	#index := #index + 1;
	//++++++++++++++++++++++++++++++++++++++++++++++++++++++++++++++/*276*/
	"DB_BIBLIOTHEQUE".Mobile[#index].Nom := 'BDE10';
	"DB_BIBLIOTHEQUE".Mobile[#index].Noeud := TRUE;
	"DB_BIBLIOTHEQUE".Mobile[#index].Mob_Suiv[0] := "Index_Mobile"('BB01');
	"DB_BIBLIOTHEQUE".Mobile[#index].Mob_Suiv[1] := "Index_Mobile"('BB02');
	"DB_BIBLIOTHEQUE".Mobile[#index].Pos[0].Nom := 'DROITE';
	"DB_BIBLIOTHEQUE".Mobile[#index].Pos[0].Mob_Suiv[0] := "Index_Mobile"('BB02');
	"DB_BIBLIOTHEQUE".Mobile[#index].Pos[1].Nom := 'GAUCHE';
	"DB_BIBLIOTHEQUE".Mobile[#index].Pos[1].Mob_Suiv[0] := "Index_Mobile"('BB01');
	"Init_Tps"(#index);


	//Entrées
	"DB_BIBLIOTHEQUE".Mobile[#index].Pos[0].Entr0_Ap_Pos[0] := "I_RP_BDE10_BB1";
	"DB_BIBLIOTHEQUE".Mobile[#index].Pos[0].Entr1_Ap_Pos[0] := "I_RP_BDE10_BB2";
	// "DB_BIBLIOTHEQUE".Mobile[#index].Pos[0].Sort1[0] := "I_CP_B2DE10_BB2";
	// "DB_BIBLIOTHEQUE".Mobile[#index].Pos[0].Sort0[0] := "I_CP_B2DE10_BB1";
	// "DB_BIBLIOTHEQUE".Mobile[#index].Pos[0].Sort0_Pr_Fin_Pos[0] := "I_CP_B2DE10_BB2";
	// "DB_BIBLIOTHEQUE".Mobile[#index].Pos[0].Sort0_Pr_Fin_Pos[1] := "I_CP_B2DE10_BB1";

	"DB_BIBLIOTHEQUE".Mobile[#index].Pos[1].Entr0_Ap_Pos[1] := "I_RP_BDE10_BB2";
	"DB_BIBLIOTHEQUE".Mobile[#index].Pos[1].Entr1_Ap_Pos[0] := "I_RP_BDE10_BB1";

	//Sorties
	// "DB_BIBLIOTHEQUE".Mobile[#index].Pos[1].Sort1[0] := "I_CP_B2DE10_BB1";
	// "DB_BIBLIOTHEQUE".Mobile[#index].Pos[1].Sort0[0] := "I_CP_B2DE10_BB2";
	// "DB_BIBLIOTHEQUE".Mobile[#index].Pos[1].Sort0_Pr_Fin_Pos[0] := "I_CP_B2DE10_BB2";
	// "DB_BIBLIOTHEQUE".Mobile[#index].Pos[1].Sort0_Pr_Fin_Pos[1] := "I_CP_B2DE10_BB1";
	#index := #index + 1;
	//++++++++++++++++++++++++++++++++++++++++++++++++++++++++++++++/*277*/
	"DB_BIBLIOTHEQUE".Mobile[#index].Nom := 'E11';
	"DB_BIBLIOTHEQUE".Mobile[#index].Mob_Suiv[0] := "Index_Mobile"('BDE11');
	"DB_BIBLIOTHEQUE".Mobile[#index].Pos[0].Nom := 'DROIT';
	"DB_BIBLIOTHEQUE".Mobile[#index].Pos[0].Mob_Suiv[0] := "Index_Mobile"('BDE11');
	"Init_Tps"(#index);

	// Entrées avant pos
	"DB_BIBLIOTHEQUE".Mobile[#index].Pos[0].Entr0_Av_Pos[0] := "I_RD_DISJ_E11";
	"DB_BIBLIOTHEQUE".Mobile[#index].Pos[0].Entr0_Av_Pos[1] := "I_RD_DBHG_E11";
	"DB_BIBLIOTHEQUE".Mobile[#index].Pos[0].Entr0_Av_Pos[2] := "I_RD_DBHD_E11";
	"DB_BIBLIOTHEQUE".Mobile[#index].Pos[0].Entr0_Av_Pos[3] := "I_RD_DBBG_E11";
	"DB_BIBLIOTHEQUE".Mobile[#index].Pos[0].Entr0_Av_Pos[4] := "I_RD_DBBD_E11";
	// Entrées apres pos
	"DB_BIBLIOTHEQUE".Mobile[#index].Pos[0].Entr0_Ap_Pos[0] := "I_RD_DISJ_E11";
	"DB_BIBLIOTHEQUE".Mobile[#index].Pos[0].Entr0_Ap_Pos[1] := "I_RD_DBHG_E11";
	"DB_BIBLIOTHEQUE".Mobile[#index].Pos[0].Entr0_Ap_Pos[2] := "I_RD_DBHD_E11";
	"DB_BIBLIOTHEQUE".Mobile[#index].Pos[0].Entr0_Ap_Pos[3] := "I_RD_DBBG_E11";
	"DB_BIBLIOTHEQUE".Mobile[#index].Pos[0].Entr0_Ap_Pos[4] := "I_RD_DBBD_E11";

	"DB_BIBLIOTHEQUE".Mobile[#index].Pos[0].Entr1_Ap_Pos[0] := "I_RR_E11";
	"DB_BIBLIOTHEQUE".Mobile[#index].Pos[0].Entr1_Ap_Pos[1] := "I_RM_E11";


	// Entrées fin pos
	"DB_BIBLIOTHEQUE".Mobile[#index].Pos[0].Entr0_Ap_Fin_Pos[0] := "I_RM_E11";

	// Sorties
	"DB_BIBLIOTHEQUE".Mobile[#index].Pos[0].Sort1[0] := "I_CM_E11";
	"DB_BIBLIOTHEQUE".Mobile[#index].Pos[0].Sort0_Pr_Fin_Pos[0] := "I_CM_E11";
	#index := #index + 1;
	//++++++++++++++++++++++++++++++++++++++++++++++++++++++++++++++/*278*/
	"DB_BIBLIOTHEQUE".Mobile[#index].Nom := 'BDE11';
	"DB_BIBLIOTHEQUE".Mobile[#index].Noeud := TRUE;
	"DB_BIBLIOTHEQUE".Mobile[#index].Mob_Suiv[0] := "Index_Mobile"('TMEL');
	"DB_BIBLIOTHEQUE".Mobile[#index].Mob_Suiv[1] := "Index_Mobile"('TMEL2');
	"DB_BIBLIOTHEQUE".Mobile[#index].Pos[0].Nom := 'DROITE';
	"DB_BIBLIOTHEQUE".Mobile[#index].Pos[0].Mob_Suiv[0] := "Index_Mobile"('TMEL');
	"DB_BIBLIOTHEQUE".Mobile[#index].Pos[1].Nom := 'GAUCHE';
	"DB_BIBLIOTHEQUE".Mobile[#index].Pos[1].Mob_Suiv[0] := "Index_Mobile"('TMEL2');


	"Init_Tps"(#index);

	//Entrées
	"DB_BIBLIOTHEQUE".Mobile[#index].Pos[0].Entr0_Ap_Pos[0] := "I_RP_BDE11_TMEL2";
	"DB_BIBLIOTHEQUE".Mobile[#index].Pos[0].Entr1_Ap_Pos[0] := "I_RP_BDE11_TMEL1";
	"DB_BIBLIOTHEQUE".Mobile[#index].Pos[0].Sort1[0] := "I_CP_BDE11_TMEL1";
	"DB_BIBLIOTHEQUE".Mobile[#index].Pos[0].Sort0[0] := "I_CP_BDE11_TMEL2";
	"DB_BIBLIOTHEQUE".Mobile[#index].Pos[0].Sort0_Pr_Fin_Pos[0] := "I_CP_BDE11_TMEL1";
	"DB_BIBLIOTHEQUE".Mobile[#index].Pos[0].Sort0_Pr_Fin_Pos[1] := "I_CP_BDE11_TMEL2";


	"DB_BIBLIOTHEQUE".Mobile[#index].Pos[1].Entr0_Ap_Pos[1] := "I_RP_BDE11_TMEL1";
	"DB_BIBLIOTHEQUE".Mobile[#index].Pos[1].Entr1_Ap_Pos[0] := "I_RP_BDE11_TMEL2";

	//Sorties
	"DB_BIBLIOTHEQUE".Mobile[#index].Pos[1].Sort1[0] := "I_CP_BDE11_TMEL2";
	"DB_BIBLIOTHEQUE".Mobile[#index].Pos[1].Sort0[0] := "I_CP_BDE11_TMEL1";
	"DB_BIBLIOTHEQUE".Mobile[#index].Pos[1].Sort0_Pr_Fin_Pos[0] := "I_CP_BDE11_TMEL1";
	"DB_BIBLIOTHEQUE".Mobile[#index].Pos[1].Sort0_Pr_Fin_Pos[1] := "I_CP_BDE11_TMEL2";
	#index := #index + 1;
	//++++++++++++++++++++++++++++++++++++++++++++++++++++++++++++++/*279*/
	"DB_BIBLIOTHEQUE".Mobile[#index].Nom := 'E30';
	"DB_BIBLIOTHEQUE".Mobile[#index].Mob_Suiv[0] := "Index_Mobile"('T20');
	"DB_BIBLIOTHEQUE".Mobile[#index].Pos[0].Nom := 'MARCHE';
	"DB_BIBLIOTHEQUE".Mobile[#index].Pos[0].Mob_Suiv[0] := "Index_Mobile"('T20');
	"DB_BIBLIOTHEQUE".Mobile[#index].Tps_Asserv := t#3s;
	"DB_BIBLIOTHEQUE".Mobile[#index].Tps_Vid := t#3s;
	"DB_BIBLIOTHEQUE".Mobile[#index].Tps_Att := t#500ms;
	"DB_BIBLIOTHEQUE".Mobile[#index].Tps_Arr := t#0ms;
	"DB_BIBLIOTHEQUE".Mobile[#index].Tps_Max_Mar_Forc := t#5s;

	// Entrées avant pos
	"DB_BIBLIOTHEQUE".Mobile[#index].Pos[0].Entr0_Av_Pos[0] := "I_RD_DISJ_E30";
	"DB_BIBLIOTHEQUE".Mobile[#index].Pos[0].Entr0_Av_Pos[1] := "I_RD_DBHG_E30";
	"DB_BIBLIOTHEQUE".Mobile[#index].Pos[0].Entr0_Av_Pos[2] := "I_RD_DBHD_E30";
	"DB_BIBLIOTHEQUE".Mobile[#index].Pos[0].Entr0_Av_Pos[3] := "I_RD_DBBG_E30";
	"DB_BIBLIOTHEQUE".Mobile[#index].Pos[0].Entr0_Av_Pos[4] := "I_RD_DBBD_E30";
	// Entrées apres pos
	"DB_BIBLIOTHEQUE".Mobile[#index].Pos[0].Entr0_Ap_Pos[0] := "I_RD_DISJ_E30";
	"DB_BIBLIOTHEQUE".Mobile[#index].Pos[0].Entr0_Ap_Pos[1] := "I_RD_DBHG_E30";
	"DB_BIBLIOTHEQUE".Mobile[#index].Pos[0].Entr0_Ap_Pos[2] := "I_RD_DBHD_E30";
	"DB_BIBLIOTHEQUE".Mobile[#index].Pos[0].Entr0_Ap_Pos[3] := "I_RD_DBBG_E30";
	"DB_BIBLIOTHEQUE".Mobile[#index].Pos[0].Entr0_Ap_Pos[4] := "I_RD_DBBD_E30";

	// "DB_BIBLIOTHEQUE".Mobile[#index].Pos[0].Entr1_Ap_Pos[0] := "I_RR_E30";
	"DB_BIBLIOTHEQUE".Mobile[#index].Pos[0].Entr1_Ap_Pos[0] := "I_RM_E30";


	// Entrées fin pos
	//"DB_BIBLIOTHEQUE".Mobile[#index].Pos[0].Entr0_Ap_Fin_Pos[0]:="I_RM_E30";

	// Sorties
	"DB_BIBLIOTHEQUE".Mobile[#index].Pos[0].Sort1[0] := "I_CM_E30";
	"DB_BIBLIOTHEQUE".Mobile[#index].Pos[0].Sort0_Pr_Fin_Pos[0] := "I_CM_E30";
	#index := #index + 1;
	//++++++++++++++++++++++++++++++++++++++++++++++++++++++++++++++/*280*/
	"DB_BIBLIOTHEQUE".Mobile[#index].Nom := 'Ext1_BB1';
	"DB_BIBLIOTHEQUE".Mobile[#index].Pos[0].Nom := 'FERMETURE';
	"DB_BIBLIOTHEQUE".Mobile[#index].Pos[1].Nom := 'OUVERTURE';
	"DB_BIBLIOTHEQUE".Mobile[#index].Tjr_Desasservi := TRUE;
	"Init_Tps"(#index);

	//position fermeture
	"DB_BIBLIOTHEQUE".Mobile[#index].Pos[0].Entr0_Ap_Pos[0] := "I_RPO_TRBB1";
	"DB_BIBLIOTHEQUE".Mobile[#index].Pos[0].Entr1_Ap_Pos[0] := "I_RPF_TRBB1";
	"DB_BIBLIOTHEQUE".Mobile[#index].Pos[0].Sort0[0] := "I_CO_TRBB1";
	"DB_BIBLIOTHEQUE".Mobile[#index].Pos[0].Sort0_Pr_Fin_Pos[0] := "I_CO_TRBB1";

	//position ouverture
	"DB_BIBLIOTHEQUE".Mobile[#index].Pos[1].Entr0_Ap_Pos[0] := "I_RPF_TRBB1";
	"DB_BIBLIOTHEQUE".Mobile[#index].Pos[1].Entr1_Ap_Pos[0] := "I_RPO_TRBB1";
	"DB_BIBLIOTHEQUE".Mobile[#index].Pos[1].Sort1[0] := "I_CO_TRBB1";
	"DB_BIBLIOTHEQUE".Mobile[#index].Pos[1].Sort0_Pr_Fin_Pos[0] := "I_CO_TRBB1";
	#index := #index + 1;
	//++++++++++++++++++++++++++++++++++++++++++++++++++++++++++++++/*281*/
	"DB_BIBLIOTHEQUE".Mobile[#index].Nom := 'Ext1_BB2';
	"DB_BIBLIOTHEQUE".Mobile[#index].Pos[0].Nom := 'FERMETURE';
	"DB_BIBLIOTHEQUE".Mobile[#index].Pos[1].Nom := 'OUVERTURE';
	"DB_BIBLIOTHEQUE".Mobile[#index].Tjr_Desasservi := TRUE;
	"Init_Tps"(#index);

	//position fermeture
	"DB_BIBLIOTHEQUE".Mobile[#index].Pos[0].Entr0_Ap_Pos[0] := "I_RPO_TRBB2";
	"DB_BIBLIOTHEQUE".Mobile[#index].Pos[0].Entr1_Ap_Pos[0] := "I_RPF_TRBB2";
	"DB_BIBLIOTHEQUE".Mobile[#index].Pos[0].Sort0[0] := "I_CO_TRBB2";
	"DB_BIBLIOTHEQUE".Mobile[#index].Pos[0].Sort0_Pr_Fin_Pos[0] := "I_CO_TRBB2";

	//position ouverture
	"DB_BIBLIOTHEQUE".Mobile[#index].Pos[1].Entr0_Ap_Pos[0] := "I_RPF_TRBB2";
	"DB_BIBLIOTHEQUE".Mobile[#index].Pos[1].Entr1_Ap_Pos[0] := "I_RPO_TRBB2";
	"DB_BIBLIOTHEQUE".Mobile[#index].Pos[1].Sort1[0] := "I_CO_TRBB2";
	"DB_BIBLIOTHEQUE".Mobile[#index].Pos[1].Sort0_Pr_Fin_Pos[0] := "I_CO_TRBB2";
	#index := #index + 1;
	//++++++++++++++++++++++++++++++++++++++++++++++++++++++++++++++/*282*/
	"DB_BIBLIOTHEQUE".Mobile[#index].Nom := 'Ext1_S50';
	"DB_BIBLIOTHEQUE".Mobile[#index].Mob_Suiv[0] := "Index_Mobile"('EXT2_S50');
	"Init_Tps"(#index);

	// Position PV
	"DB_BIBLIOTHEQUE".Mobile[#index].Pos[0].Nom := 'MARCHE_PV';
	"DB_BIBLIOTHEQUE".Mobile[#index].Pos[0].Mob_Suiv[0] := "Index_Mobile"('EXT2_S50');
	"DB_BIBLIOTHEQUE".Mobile[#index].Pos[0].Suiv_Enc := "Index_Mobile"('EXT2_S50');

	// Entrées avant pos
	"DB_BIBLIOTHEQUE".Mobile[#index].Pos[0].Entr0_Av_Pos[0] := "I_RD_DISJ_EXT1_S50";
	// "DB_BIBLIOTHEQUE".Mobile[#index].Pos[0].Entr0_Av_Pos[1] := "I_RD_VFD_BP4";

	// Entrées apres pos
	"DB_BIBLIOTHEQUE".Mobile[#index].Pos[0].Entr0_Ap_Pos[1] := "I_RD_DISJ_EXT1_S50";
	//"DB_BIBLIOTHEQUE".Mobile[#index].Pos[0].Entr0_Ap_Pos[2] := "I_RD_VFD_BP4";
	//"DB_BIBLIOTHEQUE".Mobile[#index].Pos[0].Entr1_Ap_Pos[0] := "I_RR_EXT1_S50";
	"DB_BIBLIOTHEQUE".Mobile[#index].Pos[0].Entr1_Ap_Pos[0] := "I_RM_EXT1_S50";

	// Entrées fin pos
	"DB_BIBLIOTHEQUE".Mobile[#index].Pos[0].Entr0_Ap_Fin_Pos[0] := "I_RM_EXT1_S50";

	// Sorties
	"DB_BIBLIOTHEQUE".Mobile[#index].Pos[0].Sort1[0] := "I_CM_EXT1_S50";
	"DB_BIBLIOTHEQUE".Mobile[#index].Pos[0].Sort1[1] := "I_CPV_SBP4";
	"DB_BIBLIOTHEQUE".Mobile[#index].Pos[0].Sort0_Pr_Fin_Pos[0] := "I_CM_EXT1_S50";
	"DB_BIBLIOTHEQUE".Mobile[#index].Pos[0].Sort0_Pr_Fin_Pos[1] := "I_CPV_SBP4";

	// Position GV
	"DB_BIBLIOTHEQUE".Mobile[#index].Pos[1].Nom := 'MARCHE_GV';
	"DB_BIBLIOTHEQUE".Mobile[#index].Pos[1].Mob_Suiv[0] := "Index_Mobile"('EXT2_S50');
	"DB_BIBLIOTHEQUE".Mobile[#index].Pos[1].Suiv_Enc := "Index_Mobile"('EXT2_S50');

	// Entrées avant pos
	"DB_BIBLIOTHEQUE".Mobile[#index].Pos[1].Entr0_Av_Pos[0] := "I_RD_DISJ_EXT1_S50";
	// "DB_BIBLIOTHEQUE".Mobile[#index].Pos[0].Entr0_Av_Pos[1] := "I_RD_VFD_BP4";

	// Entrées apres pos
	"DB_BIBLIOTHEQUE".Mobile[#index].Pos[1].Entr0_Ap_Pos[1] := "I_RD_DISJ_EXT1_S50";
	//"DB_BIBLIOTHEQUE".Mobile[#index].Pos[0].Entr0_Ap_Pos[2] := "I_RD_VFD_BP4";
	//"DB_BIBLIOTHEQUE".Mobile[#index].Pos[0].Entr1_Ap_Pos[0] := "I_RR_EXT1_S50";
	"DB_BIBLIOTHEQUE".Mobile[#index].Pos[1].Entr1_Ap_Pos[0] := "I_RM_EXT1_S50";

	// Entrées fin pos
	"DB_BIBLIOTHEQUE".Mobile[#index].Pos[1].Entr0_Ap_Fin_Pos[0] := "I_RM_EXT1_S50";

	// Sorties
	"DB_BIBLIOTHEQUE".Mobile[#index].Pos[1].Sort1[0] := "I_CM_EXT1_S50";
	"DB_BIBLIOTHEQUE".Mobile[#index].Pos[1].Sort1[1] := "I_CGV_SBP4";
	"DB_BIBLIOTHEQUE".Mobile[#index].Pos[1].Sort0_Pr_Fin_Pos[0] := "I_CM_EXT1_S50";
	"DB_BIBLIOTHEQUE".Mobile[#index].Pos[1].Sort0_Pr_Fin_Pos[1] := "I_CGV_SBP4";
	#index := #index + 1;
	//++++++++++++++++++++++++++++++++++++++++++++++++++++++++++++++/*283*/
	"DB_BIBLIOTHEQUE".Mobile[#index].Nom := 'Ext1_S51';
	"DB_BIBLIOTHEQUE".Mobile[#index].Mob_Suiv[0] := "Index_Mobile"('EXT2_S51');
	"Init_Tps"(#index);

	// Position PV
	"DB_BIBLIOTHEQUE".Mobile[#index].Pos[0].Nom := 'MARCHE_PV';
	"DB_BIBLIOTHEQUE".Mobile[#index].Pos[0].Mob_Suiv[0] := "Index_Mobile"('EXT2_S51');
	"DB_BIBLIOTHEQUE".Mobile[#index].Pos[0].Suiv_Enc := "Index_Mobile"('EXT2_S51');
	// Entrées avant pos
	"DB_BIBLIOTHEQUE".Mobile[#index].Pos[0].Entr0_Av_Pos[0] := "I_RD_DISJ_EXT1_S51";
	//"DB_BIBLIOTHEQUE".Mobile[#index].Pos[0].Entr0_Av_Pos[1] := "I_RD_VFD_BP4";

	// Entrées apres pos
	"DB_BIBLIOTHEQUE".Mobile[#index].Pos[0].Entr0_Ap_Pos[1] := "I_RD_DISJ_EXT1_S51";
	//"DB_BIBLIOTHEQUE".Mobile[#index].Pos[0].Entr0_Ap_Pos[2] := "I_RD_VFD_BP4";
	//"DB_BIBLIOTHEQUE".Mobile[#index].Pos[0].Entr1_Ap_Pos[0] := "I_RR_EXT1_S51";
	"DB_BIBLIOTHEQUE".Mobile[#index].Pos[0].Entr1_Ap_Pos[0] := "I_RM_EXT1_S51";

	// Entrées fin pos
	"DB_BIBLIOTHEQUE".Mobile[#index].Pos[0].Entr0_Ap_Fin_Pos[0] := "I_RM_EXT1_S51";

	// Sorties
	"DB_BIBLIOTHEQUE".Mobile[#index].Pos[0].Sort1[0] := "I_CM_EXT1_S51";
	"DB_BIBLIOTHEQUE".Mobile[#index].Pos[0].Sort1[1] := "I_CPV_SBP4";
	"DB_BIBLIOTHEQUE".Mobile[#index].Pos[0].Sort0_Pr_Fin_Pos[0] := "I_CM_EXT1_S51";
	"DB_BIBLIOTHEQUE".Mobile[#index].Pos[0].Sort0_Pr_Fin_Pos[1] := "I_CPV_SBP4";

	// Position GV
	"DB_BIBLIOTHEQUE".Mobile[#index].Pos[1].Nom := 'MARCHE_GV';
	"DB_BIBLIOTHEQUE".Mobile[#index].Pos[1].Mob_Suiv[0] := "Index_Mobile"('EXT2_S51');
	"DB_BIBLIOTHEQUE".Mobile[#index].Pos[1].Suiv_Enc := "Index_Mobile"('EXT2_S51');
	// Entrées avant pos
	"DB_BIBLIOTHEQUE".Mobile[#index].Pos[1].Entr0_Av_Pos[0] := "I_RD_DISJ_EXT1_S51";
	//"DB_BIBLIOTHEQUE".Mobile[#index].Pos[0].Entr0_Av_Pos[1] := "I_RD_VFD_BP4";

	// Entrées apres pos
	"DB_BIBLIOTHEQUE".Mobile[#index].Pos[1].Entr0_Ap_Pos[1] := "I_RD_DISJ_EXT1_S51";
	//"DB_BIBLIOTHEQUE".Mobile[#index].Pos[0].Entr0_Ap_Pos[2] := "I_RD_VFD_BP4";
	//"DB_BIBLIOTHEQUE".Mobile[#index].Pos[0].Entr1_Ap_Pos[0] := "I_RR_EXT1_S51";
	"DB_BIBLIOTHEQUE".Mobile[#index].Pos[1].Entr1_Ap_Pos[0] := "I_RM_EXT1_S51";

	// Entrées fin pos
	"DB_BIBLIOTHEQUE".Mobile[#index].Pos[1].Entr0_Ap_Fin_Pos[0] := "I_RM_EXT1_S51";

	// Sorties
	"DB_BIBLIOTHEQUE".Mobile[#index].Pos[1].Sort1[0] := "I_CM_EXT1_S51";
	"DB_BIBLIOTHEQUE".Mobile[#index].Pos[1].Sort1[1] := "I_CGV_SBP4";
	"DB_BIBLIOTHEQUE".Mobile[#index].Pos[1].Sort0_Pr_Fin_Pos[0] := "I_CM_EXT1_S51";
	"DB_BIBLIOTHEQUE".Mobile[#index].Pos[1].Sort0_Pr_Fin_Pos[1] := "I_CGV_SBP4";
	#index := #index + 1;
	//++++++++++++++++++++++++++++++++++++++++++++++++++++++++++++++/*284*/
	"DB_BIBLIOTHEQUE".Mobile[#index].Nom := 'Ext1_S52';
	"DB_BIBLIOTHEQUE".Mobile[#index].Mob_Suiv[0] := "Index_Mobile"('EXT2_S52');
	"Init_Tps"(#index);

	// Position PV
	"DB_BIBLIOTHEQUE".Mobile[#index].Pos[0].Nom := 'MARCHE_PV';
	"DB_BIBLIOTHEQUE".Mobile[#index].Pos[0].Mob_Suiv[0] := "Index_Mobile"('EXT2_S52');
	"DB_BIBLIOTHEQUE".Mobile[#index].Pos[0].Suiv_Enc := "Index_Mobile"('EXT2_S52');
	// Entrées avant pos
	"DB_BIBLIOTHEQUE".Mobile[#index].Pos[0].Entr0_Av_Pos[0] := "I_RD_DISJ_EXT1_S52";
	//"DB_BIBLIOTHEQUE".Mobile[#index].Pos[0].Entr0_Av_Pos[1] := "I_RD_VFD_BP4";
	// Entrées apres pos

	"DB_BIBLIOTHEQUE".Mobile[#index].Pos[0].Entr0_Ap_Pos[1] := "I_RD_DISJ_EXT1_S52";
	//"DB_BIBLIOTHEQUE".Mobile[#index].Pos[0].Entr0_Ap_Pos[2] := "I_RD_VFD_BP4";

	//"DB_BIBLIOTHEQUE".Mobile[#index].Pos[0].Entr1_Ap_Pos[0] := "I_RR_EXT1_S52";
	"DB_BIBLIOTHEQUE".Mobile[#index].Pos[0].Entr1_Ap_Pos[0] := "I_RM_EXT1_S52";

	// Entrées fin pos
	"DB_BIBLIOTHEQUE".Mobile[#index].Pos[0].Entr0_Ap_Fin_Pos[0] := "I_RM_EXT1_S52";

	// Sorties
	"DB_BIBLIOTHEQUE".Mobile[#index].Pos[0].Sort1[0] := "I_CM_EXT1_S52";
	"DB_BIBLIOTHEQUE".Mobile[#index].Pos[0].Sort1[1] := "I_CPV_SBP4";
	"DB_BIBLIOTHEQUE".Mobile[#index].Pos[0].Sort0_Pr_Fin_Pos[0] := "I_CM_EXT1_S52";
	"DB_BIBLIOTHEQUE".Mobile[#index].Pos[0].Sort0_Pr_Fin_Pos[1] := "I_CPV_SBP4";

	// Position GV
	"DB_BIBLIOTHEQUE".Mobile[#index].Pos[1].Nom := 'MARCHE_GV';
	"DB_BIBLIOTHEQUE".Mobile[#index].Pos[1].Mob_Suiv[0] := "Index_Mobile"('EXT2_S52');
	"DB_BIBLIOTHEQUE".Mobile[#index].Pos[1].Suiv_Enc := "Index_Mobile"('EXT2_S52');
	// Entrées avant pos
	"DB_BIBLIOTHEQUE".Mobile[#index].Pos[1].Entr0_Av_Pos[0] := "I_RD_DISJ_EXT1_S52";
	//"DB_BIBLIOTHEQUE".Mobile[#index].Pos[0].Entr0_Av_Pos[1] := "I_RD_VFD_BP4";
	// Entrées apres pos

	"DB_BIBLIOTHEQUE".Mobile[#index].Pos[1].Entr0_Ap_Pos[1] := "I_RD_DISJ_EXT1_S52";
	//"DB_BIBLIOTHEQUE".Mobile[#index].Pos[0].Entr0_Ap_Pos[2] := "I_RD_VFD_BP4";

	//"DB_BIBLIOTHEQUE".Mobile[#index].Pos[0].Entr1_Ap_Pos[0] := "I_RR_EXT1_S52";
	"DB_BIBLIOTHEQUE".Mobile[#index].Pos[1].Entr1_Ap_Pos[0] := "I_RM_EXT1_S52";

	// Entrées fin pos
	"DB_BIBLIOTHEQUE".Mobile[#index].Pos[1].Entr0_Ap_Fin_Pos[0] := "I_RM_EXT1_S52";

	// Sorties
	"DB_BIBLIOTHEQUE".Mobile[#index].Pos[1].Sort1[0] := "I_CM_EXT1_S52";
	"DB_BIBLIOTHEQUE".Mobile[#index].Pos[1].Sort1[1] := "I_CGV_SBP4";
	"DB_BIBLIOTHEQUE".Mobile[#index].Pos[1].Sort0_Pr_Fin_Pos[0] := "I_CM_EXT1_S52";
	"DB_BIBLIOTHEQUE".Mobile[#index].Pos[1].Sort0_Pr_Fin_Pos[1] := "I_CGV_SBP4";
	#index := #index + 1;
	//++++++++++++++++++++++++++++++++++++++++++++++++++++++++++++++/*285*/
	"DB_BIBLIOTHEQUE".Mobile[#index].Nom := 'Ext1_S53';
	"DB_BIBLIOTHEQUE".Mobile[#index].Mob_Suiv[0] := "Index_Mobile"('EXT2_S53');
	"Init_Tps"(#index);

	// Position PV
	"DB_BIBLIOTHEQUE".Mobile[#index].Pos[0].Nom := 'MARCHE_PV';
	"DB_BIBLIOTHEQUE".Mobile[#index].Pos[0].Mob_Suiv[0] := "Index_Mobile"('EXT2_S53');
	"DB_BIBLIOTHEQUE".Mobile[#index].Pos[0].Suiv_Enc := "Index_Mobile"('EXT2_S53');

	// Entrées avant pos
	"DB_BIBLIOTHEQUE".Mobile[#index].Pos[0].Entr0_Av_Pos[0] := "I_RD_DISJ_EXT1_S53";
	//"DB_BIBLIOTHEQUE".Mobile[#index].Pos[0].Entr0_Av_Pos[1] := "I_RD_VFD_BP4";

	// Entrées apres pos
	"DB_BIBLIOTHEQUE".Mobile[#index].Pos[0].Entr0_Ap_Pos[1] := "I_RD_DISJ_EXT1_S53";
	//"DB_BIBLIOTHEQUE".Mobile[#index].Pos[0].Entr0_Ap_Pos[2] := "I_RD_VFD_BP4";
	//"DB_BIBLIOTHEQUE".Mobile[#index].Pos[0].Entr1_Ap_Pos[0] := "I_RR_EXT1_S53";
	"DB_BIBLIOTHEQUE".Mobile[#index].Pos[0].Entr1_Ap_Pos[0] := "I_RM_EXT1_S53";

	// Entrées fin pos
	"DB_BIBLIOTHEQUE".Mobile[#index].Pos[0].Entr0_Ap_Fin_Pos[0] := "I_RM_EXT1_S53";

	// Sorties
	"DB_BIBLIOTHEQUE".Mobile[#index].Pos[0].Sort1[0] := "I_CM_EXT1_S53";
	"DB_BIBLIOTHEQUE".Mobile[#index].Pos[0].Sort1[1] := "I_CPV_SBP4";
	"DB_BIBLIOTHEQUE".Mobile[#index].Pos[0].Sort0_Pr_Fin_Pos[0] := "I_CM_EXT1_S53";
	"DB_BIBLIOTHEQUE".Mobile[#index].Pos[0].Sort0_Pr_Fin_Pos[1] := "I_CPV_SBP4";

	// Position GV
	"DB_BIBLIOTHEQUE".Mobile[#index].Pos[1].Nom := 'MARCHE_GV';
	"DB_BIBLIOTHEQUE".Mobile[#index].Pos[1].Mob_Suiv[0] := "Index_Mobile"('EXT2_S53');
	"DB_BIBLIOTHEQUE".Mobile[#index].Pos[1].Suiv_Enc := "Index_Mobile"('EXT2_S53');
	// Entrées avant pos
	"DB_BIBLIOTHEQUE".Mobile[#index].Pos[1].Entr0_Av_Pos[0] := "I_RD_DISJ_EXT1_S53";
	//"DB_BIBLIOTHEQUE".Mobile[#index].Pos[0].Entr0_Av_Pos[1] := "I_RD_VFD_BP4";

	// Entrées apres pos
	"DB_BIBLIOTHEQUE".Mobile[#index].Pos[1].Entr0_Ap_Pos[1] := "I_RD_DISJ_EXT1_S53";
	//"DB_BIBLIOTHEQUE".Mobile[#index].Pos[0].Entr0_Ap_Pos[2] := "I_RD_VFD_BP4";
	//"DB_BIBLIOTHEQUE".Mobile[#index].Pos[0].Entr1_Ap_Pos[0] := "I_RR_EXT1_S53";
	"DB_BIBLIOTHEQUE".Mobile[#index].Pos[1].Entr1_Ap_Pos[0] := "I_RM_EXT1_S53";

	// Entrées fin pos
	"DB_BIBLIOTHEQUE".Mobile[#index].Pos[1].Entr0_Ap_Fin_Pos[0] := "I_RM_EXT1_S53";

	// Sorties
	"DB_BIBLIOTHEQUE".Mobile[#index].Pos[1].Sort1[0] := "I_CM_EXT1_S53";
	"DB_BIBLIOTHEQUE".Mobile[#index].Pos[1].Sort1[1] := "I_CGV_SBP4";
	"DB_BIBLIOTHEQUE".Mobile[#index].Pos[1].Sort0_Pr_Fin_Pos[0] := "I_CM_EXT1_S53";
	"DB_BIBLIOTHEQUE".Mobile[#index].Pos[1].Sort0_Pr_Fin_Pos[1] := "I_CGV_SBP4";
	#index := #index + 1;
	//++++++++++++++++++++++++++++++++++++++++++++++++++++++++++++++/*286*/
	"DB_BIBLIOTHEQUE".Mobile[#index].Nom := 'Ext1_S54';
	"DB_BIBLIOTHEQUE".Mobile[#index].Mob_Suiv[0] := "Index_Mobile"('EXT2_S54');
	"Init_Tps"(#index);

	// Position PV
	"DB_BIBLIOTHEQUE".Mobile[#index].Pos[0].Nom := 'MARCHE_PV';
	"DB_BIBLIOTHEQUE".Mobile[#index].Pos[0].Mob_Suiv[0] := "Index_Mobile"('EXT2_S54');
	"DB_BIBLIOTHEQUE".Mobile[#index].Pos[0].Suiv_Enc := "Index_Mobile"('EXT2_S54');

	// Entrées avant pos
	"DB_BIBLIOTHEQUE".Mobile[#index].Pos[0].Entr0_Av_Pos[0] := "I_RD_DISJ_EXT1_S54";
	//"DB_BIBLIOTHEQUE".Mobile[#index].Pos[0].Entr0_Av_Pos[1] := "I_RD_VFD_BP4";

	// Entrées apres pos
	"DB_BIBLIOTHEQUE".Mobile[#index].Pos[0].Entr0_Ap_Pos[1] := "I_RD_DISJ_EXT1_S54";
	//"DB_BIBLIOTHEQUE".Mobile[#index].Pos[0].Entr0_Ap_Pos[2] := "I_RD_VFD_BP4";
	//"DB_BIBLIOTHEQUE".Mobile[#index].Pos[0].Entr1_Ap_Pos[0] := "I_RR_EXT1_S54";
	"DB_BIBLIOTHEQUE".Mobile[#index].Pos[0].Entr1_Ap_Pos[0] := "I_RM_EXT1_S54";

	// Entrées fin pos
	"DB_BIBLIOTHEQUE".Mobile[#index].Pos[0].Entr0_Ap_Fin_Pos[0] := "I_RM_EXT1_S54";

	// Sorties
	"DB_BIBLIOTHEQUE".Mobile[#index].Pos[0].Sort1[0] := "I_CM_EXT1_S54";
	"DB_BIBLIOTHEQUE".Mobile[#index].Pos[0].Sort1[1] := "I_CPV_SBP4";
	"DB_BIBLIOTHEQUE".Mobile[#index].Pos[0].Sort0_Pr_Fin_Pos[0] := "I_CM_EXT1_S54";
	"DB_BIBLIOTHEQUE".Mobile[#index].Pos[0].Sort0_Pr_Fin_Pos[1] := "I_CPV_SBP4";

	// Position GV
	"DB_BIBLIOTHEQUE".Mobile[#index].Pos[1].Nom := 'MARCHE_GV';
	"DB_BIBLIOTHEQUE".Mobile[#index].Pos[1].Mob_Suiv[0] := "Index_Mobile"('EXT2_S54');
	"DB_BIBLIOTHEQUE".Mobile[#index].Pos[1].Suiv_Enc := "Index_Mobile"('EXT2_S54');
	// Entrées avant pos
	"DB_BIBLIOTHEQUE".Mobile[#index].Pos[1].Entr0_Av_Pos[0] := "I_RD_DISJ_EXT1_S54";
	//"DB_BIBLIOTHEQUE".Mobile[#index].Pos[0].Entr0_Av_Pos[1] := "I_RD_VFD_BP4";

	// Entrées apres pos
	"DB_BIBLIOTHEQUE".Mobile[#index].Pos[1].Entr0_Ap_Pos[1] := "I_RD_DISJ_EXT1_S54";
	//"DB_BIBLIOTHEQUE".Mobile[#index].Pos[0].Entr0_Ap_Pos[2] := "I_RD_VFD_BP4";
	//"DB_BIBLIOTHEQUE".Mobile[#index].Pos[0].Entr1_Ap_Pos[0] := "I_RR_EXT1_S54";
	"DB_BIBLIOTHEQUE".Mobile[#index].Pos[1].Entr1_Ap_Pos[0] := "I_RM_EXT1_S54";

	// Entrées fin pos
	"DB_BIBLIOTHEQUE".Mobile[#index].Pos[1].Entr0_Ap_Fin_Pos[0] := "I_RM_EXT1_S54";

	// Sorties
	"DB_BIBLIOTHEQUE".Mobile[#index].Pos[1].Sort1[0] := "I_CM_EXT1_S54";
	"DB_BIBLIOTHEQUE".Mobile[#index].Pos[1].Sort1[1] := "I_CGV_SBP4";
	"DB_BIBLIOTHEQUE".Mobile[#index].Pos[1].Sort0_Pr_Fin_Pos[0] := "I_CM_EXT1_S54";
	"DB_BIBLIOTHEQUE".Mobile[#index].Pos[1].Sort0_Pr_Fin_Pos[1] := "I_CGV_SBP4";
	#index := #index + 1;
	//++++++++++++++++++++++++++++++++++++++++++++++++++++++++++++++/*287*/
	"DB_BIBLIOTHEQUE".Mobile[#index].Nom := 'Ext1_S55';
	"DB_BIBLIOTHEQUE".Mobile[#index].Mob_Suiv[0] := "Index_Mobile"('EXT2_S55');
	"Init_Tps"(#index);

	// Position PV
	"DB_BIBLIOTHEQUE".Mobile[#index].Pos[0].Nom := 'MARCHE_PV';
	"DB_BIBLIOTHEQUE".Mobile[#index].Pos[0].Mob_Suiv[0] := "Index_Mobile"('EXT2_S55');
	"DB_BIBLIOTHEQUE".Mobile[#index].Pos[0].Suiv_Enc := "Index_Mobile"('EXT2_S55');
	// Entrées avant pos
	"DB_BIBLIOTHEQUE".Mobile[#index].Pos[0].Entr0_Av_Pos[0] := "I_RD_DISJ_EXT1_S55";
	//"DB_BIBLIOTHEQUE".Mobile[#index].Pos[0].Entr0_Av_Pos[1] := "I_RD_VFD_BP4";

	// Entrées apres pos
	"DB_BIBLIOTHEQUE".Mobile[#index].Pos[0].Entr0_Ap_Pos[1] := "I_RD_DISJ_EXT1_S55";
	// "DB_BIBLIOTHEQUE".Mobile[#index].Pos[0].Entr0_Ap_Pos[2] := "I_RD_VFD_BP4";
	// "DB_BIBLIOTHEQUE".Mobile[#index].Pos[0].Entr1_Ap_Pos[0] := "I_RR_EXT1_S55";
	"DB_BIBLIOTHEQUE".Mobile[#index].Pos[0].Entr1_Ap_Pos[0] := "I_RM_EXT1_S55";

	// Entrées fin pos
	"DB_BIBLIOTHEQUE".Mobile[#index].Pos[0].Entr0_Ap_Fin_Pos[0] := "I_RM_EXT1_S55";

	// Sorties
	"DB_BIBLIOTHEQUE".Mobile[#index].Pos[0].Sort1[0] := "I_CM_EXT1_S55";
	"DB_BIBLIOTHEQUE".Mobile[#index].Pos[0].Sort1[1] := "I_CPV_SBP4";
	"DB_BIBLIOTHEQUE".Mobile[#index].Pos[0].Sort0_Pr_Fin_Pos[0] := "I_CM_EXT1_S55";
	"DB_BIBLIOTHEQUE".Mobile[#index].Pos[0].Sort0_Pr_Fin_Pos[1] := "I_CPV_SBP4";

	// Position GV
	"DB_BIBLIOTHEQUE".Mobile[#index].Pos[1].Nom := 'MARCHE_GV';
	"DB_BIBLIOTHEQUE".Mobile[#index].Pos[1].Mob_Suiv[0] := "Index_Mobile"('EXT2_S55');
	"DB_BIBLIOTHEQUE".Mobile[#index].Pos[1].Suiv_Enc := "Index_Mobile"('EXT2_S55');
	// Entrées avant pos
	"DB_BIBLIOTHEQUE".Mobile[#index].Pos[1].Entr0_Av_Pos[0] := "I_RD_DISJ_EXT1_S55";
	//"DB_BIBLIOTHEQUE".Mobile[#index].Pos[0].Entr0_Av_Pos[1] := "I_RD_VFD_BP4";

	// Entrées apres pos
	"DB_BIBLIOTHEQUE".Mobile[#index].Pos[1].Entr0_Ap_Pos[1] := "I_RD_DISJ_EXT1_S55";
	// "DB_BIBLIOTHEQUE".Mobile[#index].Pos[0].Entr0_Ap_Pos[2] := "I_RD_VFD_BP4";
	// "DB_BIBLIOTHEQUE".Mobile[#index].Pos[0].Entr1_Ap_Pos[0] := "I_RR_EXT1_S55";
	"DB_BIBLIOTHEQUE".Mobile[#index].Pos[1].Entr1_Ap_Pos[0] := "I_RM_EXT1_S55";

	// Entrées fin pos
	"DB_BIBLIOTHEQUE".Mobile[#index].Pos[1].Entr0_Ap_Fin_Pos[0] := "I_RM_EXT1_S55";

	// Sorties
	"DB_BIBLIOTHEQUE".Mobile[#index].Pos[1].Sort1[0] := "I_CM_EXT1_S55";
	"DB_BIBLIOTHEQUE".Mobile[#index].Pos[1].Sort1[1] := "I_CGV_SBP4";
	"DB_BIBLIOTHEQUE".Mobile[#index].Pos[1].Sort0_Pr_Fin_Pos[0] := "I_CM_EXT1_S55";
	"DB_BIBLIOTHEQUE".Mobile[#index].Pos[1].Sort0_Pr_Fin_Pos[1] := "I_CGV_SBP4";
	#index := #index + 1;
	//++++++++++++++++++++++++++++++++++++++++++++++++++++++++++++++/*288*/
	"DB_BIBLIOTHEQUE".Mobile[#index].Nom := 'Ext1_S56';
	"DB_BIBLIOTHEQUE".Mobile[#index].Mob_Suiv[0] := "Index_Mobile"('EXT2_S56');
	"Init_Tps"(#index);

	// Position PV
	"DB_BIBLIOTHEQUE".Mobile[#index].Pos[0].Nom := 'MARCHE_PV';
	"DB_BIBLIOTHEQUE".Mobile[#index].Pos[0].Mob_Suiv[0] := "Index_Mobile"('EXT2_S56');
	"DB_BIBLIOTHEQUE".Mobile[#index].Pos[0].Suiv_Enc := "Index_Mobile"('EXT2_S56');

	// Entrées avant pos
	"DB_BIBLIOTHEQUE".Mobile[#index].Pos[0].Entr0_Av_Pos[0] := "I_RD_DISJ_EXT1_S56";
	//"DB_BIBLIOTHEQUE".Mobile[#index].Pos[0].Entr0_Av_Pos[1] := "I_RD_VFD_BP4";

	// Entrées apres pos
	"DB_BIBLIOTHEQUE".Mobile[#index].Pos[0].Entr0_Ap_Pos[0] := "I_RD_DISJ_EXT1_S56";
	// "DB_BIBLIOTHEQUE".Mobile[#index].Pos[0].Entr0_Ap_Pos[2] := "I_RD_VFD_BP4";
	// "DB_BIBLIOTHEQUE".Mobile[#index].Pos[0].Entr1_Ap_Pos[0] := "I_RR_EXT1_S56";
	"DB_BIBLIOTHEQUE".Mobile[#index].Pos[0].Entr1_Ap_Pos[0] := "I_RM_EXT1_S56";

	// Entrées fin pos
	"DB_BIBLIOTHEQUE".Mobile[#index].Pos[0].Entr0_Ap_Fin_Pos[0] := "I_RM_EXT1_S56";

	// Sorties
	"DB_BIBLIOTHEQUE".Mobile[#index].Pos[0].Sort1[0] := "I_CM_EXT1_S56";
	"DB_BIBLIOTHEQUE".Mobile[#index].Pos[0].Sort1[1] := "I_CPV_SBP4";
	"DB_BIBLIOTHEQUE".Mobile[#index].Pos[0].Sort0_Pr_Fin_Pos[0] := "I_CM_EXT1_S56";
	"DB_BIBLIOTHEQUE".Mobile[#index].Pos[0].Sort0_Pr_Fin_Pos[1] := "I_CPV_SBP4";

	// Position GV
	"DB_BIBLIOTHEQUE".Mobile[#index].Pos[1].Nom := 'MARCHE_GV';
	"DB_BIBLIOTHEQUE".Mobile[#index].Pos[1].Mob_Suiv[0] := "Index_Mobile"('EXT2_S56');
	"DB_BIBLIOTHEQUE".Mobile[#index].Pos[1].Suiv_Enc := "Index_Mobile"('EXT2_S56');
	// Entrées avant pos
	"DB_BIBLIOTHEQUE".Mobile[#index].Pos[1].Entr0_Av_Pos[0] := "I_RD_DISJ_EXT1_S56";
	//"DB_BIBLIOTHEQUE".Mobile[#index].Pos[0].Entr0_Av_Pos[1] := "I_RD_VFD_BP4";

	// Entrées apres pos
	"DB_BIBLIOTHEQUE".Mobile[#index].Pos[1].Entr0_Ap_Pos[0] := "I_RD_DISJ_EXT1_S56";
	// "DB_BIBLIOTHEQUE".Mobile[#index].Pos[0].Entr0_Ap_Pos[2] := "I_RD_VFD_BP4";
	// "DB_BIBLIOTHEQUE".Mobile[#index].Pos[0].Entr1_Ap_Pos[0] := "I_RR_EXT1_S56";
	"DB_BIBLIOTHEQUE".Mobile[#index].Pos[1].Entr1_Ap_Pos[0] := "I_RM_EXT1_S56";

	// Entrées fin pos
	"DB_BIBLIOTHEQUE".Mobile[#index].Pos[1].Entr0_Ap_Fin_Pos[0] := "I_RM_EXT1_S56";

	// Sorties
	"DB_BIBLIOTHEQUE".Mobile[#index].Pos[1].Sort1[0] := "I_CM_EXT1_S56";
	"DB_BIBLIOTHEQUE".Mobile[#index].Pos[1].Sort1[1] := "I_CGV_SBP4";
	"DB_BIBLIOTHEQUE".Mobile[#index].Pos[1].Sort0_Pr_Fin_Pos[0] := "I_CM_EXT1_S56";
	"DB_BIBLIOTHEQUE".Mobile[#index].Pos[1].Sort0_Pr_Fin_Pos[1] := "I_CGV_SBP4";
	#index := #index + 1;
	//++++++++++++++++++++++++++++++++++++++++++++++++++++++++++++++/*289*/
	"DB_BIBLIOTHEQUE".Mobile[#index].Nom := 'Ext1_S57';
	"DB_BIBLIOTHEQUE".Mobile[#index].Mob_Suiv[0] := "Index_Mobile"('EXT2_S57');
	"Init_Tps"(#index);

	// Position PV
	"DB_BIBLIOTHEQUE".Mobile[#index].Pos[0].Nom := 'MARCHE_PV';
	"DB_BIBLIOTHEQUE".Mobile[#index].Pos[0].Mob_Suiv[0] := "Index_Mobile"('EXT2_S57');
	"DB_BIBLIOTHEQUE".Mobile[#index].Pos[0].Suiv_Enc := "Index_Mobile"('EXT2_S57');
	// Entrées avant pos
	"DB_BIBLIOTHEQUE".Mobile[#index].Pos[0].Entr0_Av_Pos[0] := "I_RD_DISJ_EXT1_S57";
	//"DB_BIBLIOTHEQUE".Mobile[#index].Pos[0].Entr0_Av_Pos[1] := "I_RD_VFD_BP4";

	// Entrées apres pos
	"DB_BIBLIOTHEQUE".Mobile[#index].Pos[0].Entr0_Ap_Pos[0] := "I_RD_DISJ_EXT1_S57";
	// "DB_BIBLIOTHEQUE".Mobile[#index].Pos[0].Entr0_Ap_Pos[2] := "I_RD_VFD_BP4";
	// "DB_BIBLIOTHEQUE".Mobile[#index].Pos[0].Entr1_Ap_Pos[0] := "I_RR_EXT1_S57";
	"DB_BIBLIOTHEQUE".Mobile[#index].Pos[0].Entr1_Ap_Pos[0] := "I_RM_EXT1_S57";

	// Entrées fin pos
	"DB_BIBLIOTHEQUE".Mobile[#index].Pos[0].Entr0_Ap_Fin_Pos[0] := "I_RM_EXT1_S57";

	// Sorties
	"DB_BIBLIOTHEQUE".Mobile[#index].Pos[0].Sort1[0] := "I_CM_EXT1_S57";
	"DB_BIBLIOTHEQUE".Mobile[#index].Pos[0].Sort1[1] := "I_CPV_SBP4";
	"DB_BIBLIOTHEQUE".Mobile[#index].Pos[0].Sort0_Pr_Fin_Pos[0] := "I_CM_EXT1_S57";
	"DB_BIBLIOTHEQUE".Mobile[#index].Pos[0].Sort0_Pr_Fin_Pos[1] := "I_CPV_SBP4";

	// Position GV
	"DB_BIBLIOTHEQUE".Mobile[#index].Pos[1].Nom := 'MARCHE_GV';
	"DB_BIBLIOTHEQUE".Mobile[#index].Pos[1].Mob_Suiv[0] := "Index_Mobile"('EXT2_S57');
	"DB_BIBLIOTHEQUE".Mobile[#index].Pos[1].Suiv_Enc := "Index_Mobile"('EXT2_S57');
	// Entrées avant pos
	"DB_BIBLIOTHEQUE".Mobile[#index].Pos[1].Entr0_Av_Pos[0] := "I_RD_DISJ_EXT1_S57";
	//"DB_BIBLIOTHEQUE".Mobile[#index].Pos[0].Entr0_Av_Pos[1] := "I_RD_VFD_BP4";

	// Entrées apres pos
	"DB_BIBLIOTHEQUE".Mobile[#index].Pos[1].Entr0_Ap_Pos[0] := "I_RD_DISJ_EXT1_S57";
	// "DB_BIBLIOTHEQUE".Mobile[#index].Pos[0].Entr0_Ap_Pos[2] := "I_RD_VFD_BP4";
	// "DB_BIBLIOTHEQUE".Mobile[#index].Pos[0].Entr1_Ap_Pos[0] := "I_RR_EXT1_S57";
	"DB_BIBLIOTHEQUE".Mobile[#index].Pos[1].Entr1_Ap_Pos[0] := "I_RM_EXT1_S57";

	// Entrées fin pos
	"DB_BIBLIOTHEQUE".Mobile[#index].Pos[1].Entr0_Ap_Fin_Pos[0] := "I_RM_EXT1_S57";

	// Sorties
	"DB_BIBLIOTHEQUE".Mobile[#index].Pos[1].Sort1[0] := "I_CM_EXT1_S57";
	"DB_BIBLIOTHEQUE".Mobile[#index].Pos[1].Sort1[1] := "I_CGV_SBP4";
	"DB_BIBLIOTHEQUE".Mobile[#index].Pos[1].Sort0_Pr_Fin_Pos[0] := "I_CM_EXT1_S57";
	"DB_BIBLIOTHEQUE".Mobile[#index].Pos[1].Sort0_Pr_Fin_Pos[1] := "I_CGV_SBP4";
	#index := #index + 1;
	//++++++++++++++++++++++++++++++++++++++++++++++++++++++++++++++/*290*/
	"DB_BIBLIOTHEQUE".Mobile[#index].Nom := 'Ext1_S58';
	"DB_BIBLIOTHEQUE".Mobile[#index].Mob_Suiv[0] := "Index_Mobile"('EXT2_S58');
	"Init_Tps"(#index);

	//Position PV
	"DB_BIBLIOTHEQUE".Mobile[#index].Pos[0].Nom := 'MARCHE_PV';
	"DB_BIBLIOTHEQUE".Mobile[#index].Pos[0].Mob_Suiv[0] := "Index_Mobile"('EXT2_S58');
	"DB_BIBLIOTHEQUE".Mobile[#index].Pos[0].Suiv_Enc := "Index_Mobile"('EXT2_S58');
	// Entrées avant pos
	"DB_BIBLIOTHEQUE".Mobile[#index].Pos[0].Entr0_Av_Pos[0] := "I_RD_DISJ_EXT1_S58";
	//"DB_BIBLIOTHEQUE".Mobile[#index].Pos[0].Entr0_Av_Pos[1] := "I_RD_VFD_BP4";

	// Entrées apres pos
	"DB_BIBLIOTHEQUE".Mobile[#index].Pos[0].Entr0_Ap_Pos[0] := "I_RD_DISJ_EXT1_S58";
	//"DB_BIBLIOTHEQUE".Mobile[#index].Pos[0].Entr0_Ap_Pos[2] := "I_RD_VFD_BP4";
	//"DB_BIBLIOTHEQUE".Mobile[#index].Pos[0].Entr1_Ap_Pos[0] := "I_RR_EXT1_S58";
	"DB_BIBLIOTHEQUE".Mobile[#index].Pos[0].Entr1_Ap_Pos[0] := "I_RM_EXT1_S58";

	// Entrées fin pos
	"DB_BIBLIOTHEQUE".Mobile[#index].Pos[0].Entr0_Ap_Fin_Pos[0] := "I_RM_EXT1_S58";

	// Sorties
	"DB_BIBLIOTHEQUE".Mobile[#index].Pos[0].Sort1[0] := "I_CM_EXT1_S58";
	"DB_BIBLIOTHEQUE".Mobile[#index].Pos[0].Sort1[1] := "I_CPV_SBP4";
	"DB_BIBLIOTHEQUE".Mobile[#index].Pos[0].Sort0_Pr_Fin_Pos[0] := "I_CM_EXT1_S58";
	"DB_BIBLIOTHEQUE".Mobile[#index].Pos[0].Sort0_Pr_Fin_Pos[1] := "I_CPV_SBP4";

	//Position GV
	"DB_BIBLIOTHEQUE".Mobile[#index].Pos[1].Nom := 'MARCHE_GV';
	"DB_BIBLIOTHEQUE".Mobile[#index].Pos[1].Mob_Suiv[0] := "Index_Mobile"('EXT2_S58');
	"DB_BIBLIOTHEQUE".Mobile[#index].Pos[1].Suiv_Enc := "Index_Mobile"('EXT2_S58');
	// Entrées avant pos
	"DB_BIBLIOTHEQUE".Mobile[#index].Pos[1].Entr0_Av_Pos[0] := "I_RD_DISJ_EXT1_S58";
	//"DB_BIBLIOTHEQUE".Mobile[#index].Pos[0].Entr0_Av_Pos[1] := "I_RD_VFD_BP4";

	// Entrées apres pos
	"DB_BIBLIOTHEQUE".Mobile[#index].Pos[1].Entr0_Ap_Pos[0] := "I_RD_DISJ_EXT1_S58";
	//"DB_BIBLIOTHEQUE".Mobile[#index].Pos[0].Entr0_Ap_Pos[2] := "I_RD_VFD_BP4";
	//"DB_BIBLIOTHEQUE".Mobile[#index].Pos[0].Entr1_Ap_Pos[0] := "I_RR_EXT1_S58";
	"DB_BIBLIOTHEQUE".Mobile[#index].Pos[1].Entr1_Ap_Pos[0] := "I_RM_EXT1_S58";

	// Entrées fin pos
	"DB_BIBLIOTHEQUE".Mobile[#index].Pos[1].Entr0_Ap_Fin_Pos[0] := "I_RM_EXT1_S58";

	// Sorties
	"DB_BIBLIOTHEQUE".Mobile[#index].Pos[1].Sort1[0] := "I_CM_EXT1_S58";
	"DB_BIBLIOTHEQUE".Mobile[#index].Pos[1].Sort1[1] := "I_CGV_SBP4";
	"DB_BIBLIOTHEQUE".Mobile[#index].Pos[1].Sort0_Pr_Fin_Pos[0] := "I_CM_EXT1_S58";
	"DB_BIBLIOTHEQUE".Mobile[#index].Pos[1].Sort0_Pr_Fin_Pos[1] := "I_CGV_SBP4";
	#index := #index + 1;
	//++++++++++++++++++++++++++++++++++++++++++++++++++++++++++++++/*291*/
	"DB_BIBLIOTHEQUE".Mobile[#index].Nom := 'Alim_BR2';
	"DB_BIBLIOTHEQUE".Mobile[#index].Mob_Suiv[0] := "Index_Mobile"('BR2');
	"DB_BIBLIOTHEQUE".Mobile[#index].Pos[0].Nom := 'MARCHE';
	"DB_BIBLIOTHEQUE".Mobile[#index].Pos[0].Mob_Suiv[0] := "Index_Mobile"('BR2');
	"DB_BIBLIOTHEQUE".Mobile[#index].Pos[0].Suiv_Enc := "Index_Mobile"('BR2');
	"DB_BIBLIOTHEQUE".Mobile[#index].Tps_Att := t#500ms;
	"DB_BIBLIOTHEQUE".Mobile[#index].Tps_Arr := t#0ms;

	// Entrées avant pos
	"DB_BIBLIOTHEQUE".Mobile[#index].Pos[0].Entr0_Av_Pos[0] := "I_RD_DISJ_ALIM_BR02";
	"DB_BIBLIOTHEQUE".Mobile[#index].Pos[0].Entr0_Av_Pos[1] := "I_RD_VFD_ALIM_BR02";

	// Entrées apres pos
	"DB_BIBLIOTHEQUE".Mobile[#index].Pos[0].Entr0_Ap_Pos[1] := "I_RD_DISJ_ALIM_BR02";
	"DB_BIBLIOTHEQUE".Mobile[#index].Pos[0].Entr0_Ap_Pos[2] := "I_RD_VFD_ALIM_BR02";
	// "DB_BIBLIOTHEQUE".Mobile[#index].Pos[0].Entr1_Ap_Pos[0] := "I_RR_ALIM_BR02";
	"DB_BIBLIOTHEQUE".Mobile[#index].Pos[0].Entr1_Ap_Pos[0] := "I_RM_ALIM_BR02";

	// Entrées fin pos
	"DB_BIBLIOTHEQUE".Mobile[#index].Pos[0].Entr0_Ap_Fin_Pos[0] := "I_RM_ALIM_BR02";

	// Sorties
	"DB_BIBLIOTHEQUE".Mobile[#index].Pos[0].Sort1[0] := "I_CM_ALIM_BR02";
	"DB_BIBLIOTHEQUE".Mobile[#index].Pos[0].Sort0_Pr_Fin_Pos[0] := "I_CM_ALIM_BR02";
	#index := #index + 1;
	//++++++++++++++++++++++++++++++++++++++++++++++++++++++++++++++/*292*/
	"DB_BIBLIOTHEQUE".Mobile[#index].Nom := 'VSENS_BR2';
	"DB_BIBLIOTHEQUE".Mobile[#index].Pos[0].Nom := 'FERMETURE';
	"DB_BIBLIOTHEQUE".Mobile[#index].Pos[1].Nom := 'OUVERTURE';
	"DB_BIBLIOTHEQUE".Mobile[#index].Tjr_Desasservi := TRUE;

	//position fermeture
	"DB_BIBLIOTHEQUE".Mobile[#index].Pos[0].Entr0_Ap_Pos[0] := "I_RP_AV_VOLBR02";
	"DB_BIBLIOTHEQUE".Mobile[#index].Pos[0].Entr1_Ap_Pos[0] := "I_RP_AR_VOLBR02";
	"DB_BIBLIOTHEQUE".Mobile[#index].Pos[0].Sort0[0] := "I_C_AV_VOLBR02";
	"DB_BIBLIOTHEQUE".Mobile[#index].Pos[0].Sort0_Pr_Fin_Pos[0] := "I_C_AV_VOLBR02";

	//position ouverture
	"DB_BIBLIOTHEQUE".Mobile[#index].Pos[1].Entr0_Ap_Pos[0] := "I_RP_AR_VOLBR02";
	"DB_BIBLIOTHEQUE".Mobile[#index].Pos[1].Entr1_Ap_Pos[0] := "I_RP_AV_VOLBR02";
	"DB_BIBLIOTHEQUE".Mobile[#index].Pos[1].Sort1[0] := "I_C_AV_VOLBR02";
	"DB_BIBLIOTHEQUE".Mobile[#index].Pos[1].Sort0_Pr_Fin_Pos[0] := "I_C_AV_VOLBR02";
	"Init_Tps"(#index);
	#index := #index + 1;
	//++++++++++++++++++++++++++++++++++++++++++++++++++++++++++++++/*293*/
	"DB_BIBLIOTHEQUE".Mobile[#index].Nom := 'BR2';
	"DB_BIBLIOTHEQUE".Mobile[#index].Pos[0].Nom := 'AVANT';
	"DB_BIBLIOTHEQUE".Mobile[#index].Pos[1].Nom := 'ARRIERE';
	"DB_BIBLIOTHEQUE".Mobile[#index].Tjr_Desasservi := TRUE;
	"DB_BIBLIOTHEQUE".Mobile[#index].Tps_Att := t#500ms;
	"DB_BIBLIOTHEQUE".Mobile[#index].Tps_Arr := t#0ms;

	// Entrées avant pos
	"DB_BIBLIOTHEQUE".Mobile[#index].Pos[0].Entr0_Av_Pos[0] := "I_RD_DISJ_BR02";
	"DB_BIBLIOTHEQUE".Mobile[#index].Pos[0].Entr0_Av_Pos[1] := "I_RD_VFD_BR02";

	// Entrées apres pos
	"DB_BIBLIOTHEQUE".Mobile[#index].Pos[0].Entr0_Ap_Pos[0] := "I_RD_DISJ_BR02";
	"DB_BIBLIOTHEQUE".Mobile[#index].Pos[0].Entr0_Av_Pos[1] := "I_RD_VFD_BR02";
	// "DB_BIBLIOTHEQUE".Mobile[#index].Pos[0].Entr1_Ap_Pos[0] := "I_RR_BR02";
	"DB_BIBLIOTHEQUE".Mobile[#index].Pos[0].Entr1_Ap_Pos[0] := "I_RM_AR_BR02";

	// Entrées fin pos
	"DB_BIBLIOTHEQUE".Mobile[#index].Pos[0].Entr0_Ap_Fin_Pos[0] := "I_RM_AR_BR02";

	// Sorties
	"DB_BIBLIOTHEQUE".Mobile[#index].Pos[0].Sort1[0] := "I_CM_AR_BR02";
	"DB_BIBLIOTHEQUE".Mobile[#index].Pos[0].Sort0_Pr_Fin_Pos[0] := "I_CM_AR_BR02";
	#index := #index + 1;
	//++++++++++++++++++++++++++++++++++++++++++++++++++++++++++++++/*294*/
	"DB_BIBLIOTHEQUE".Mobile[#index].Nom := 'VH_BR2';
	"DB_BIBLIOTHEQUE".Mobile[#index].Pos[0].Nom := 'AVANT';
	"DB_BIBLIOTHEQUE".Mobile[#index].Pos[1].Nom := 'ARRIERE';
	"DB_BIBLIOTHEQUE".Mobile[#index].Tjr_Desasservi := TRUE;
	"Init_Tps"(#index);

	//Entrées
	"DB_BIBLIOTHEQUE".Mobile[#index].Pos[0].Entr0_Ap_Pos[0] := "I_CMF_VAC_BR2";
	"DB_BIBLIOTHEQUE".Mobile[#index].Pos[0].Entr1_Ap_Pos[0] := "I_CMO_VAC_BR2";
	"DB_BIBLIOTHEQUE".Mobile[#index].Pos[0].Sort1[0] := "I_CMO_VAC_BR2";
	"DB_BIBLIOTHEQUE".Mobile[#index].Pos[0].Sort0[0] := "I_CMF_VAC_BR2";
	"DB_BIBLIOTHEQUE".Mobile[#index].Pos[0].Sort0_Pr_Fin_Pos[0] := "I_CMO_VAC_BR2";
	"DB_BIBLIOTHEQUE".Mobile[#index].Pos[0].Sort0_Pr_Fin_Pos[1] := "I_CMF_VAC_BR2";

	"DB_BIBLIOTHEQUE".Mobile[#index].Pos[1].Entr0_Ap_Pos[1] := "I_RPD_VAC_BR02";
	"DB_BIBLIOTHEQUE".Mobile[#index].Pos[1].Entr1_Ap_Pos[0] := "I_RPG_VAC_BR02";

	//Sorties
	"DB_BIBLIOTHEQUE".Mobile[#index].Pos[1].Sort1[0] := "I_CMF_VAC_BR2";
	"DB_BIBLIOTHEQUE".Mobile[#index].Pos[1].Sort0[0] := "I_CMO_VAC_BR2";
	"DB_BIBLIOTHEQUE".Mobile[#index].Pos[1].Sort0_Pr_Fin_Pos[0] := "I_CMO_VAC_BR2";
	"DB_BIBLIOTHEQUE".Mobile[#index].Pos[1].Sort0_Pr_Fin_Pos[1] := "I_CMF_VAC_BR2";
	#index := #index + 1;
	//++++++++++++++++++++++++++++++++++++++++++++++++++++++++++++++/*295*/
	"DB_BIBLIOTHEQUE".Mobile[#index].Nom := 'VA_BR2';
	"DB_BIBLIOTHEQUE".Mobile[#index].Pos[0].Nom := 'FERMETURE';
	"DB_BIBLIOTHEQUE".Mobile[#index].Pos[1].Nom := 'OUVERTURE';
	"DB_BIBLIOTHEQUE".Mobile[#index].Tjr_Desasservi := TRUE;
	"Init_Tps"(#index);

	//position fermeture
	"DB_BIBLIOTHEQUE".Mobile[#index].Pos[0].Entr0_Ap_Pos[0] := "I_RPO_VASP_BR02";
	"DB_BIBLIOTHEQUE".Mobile[#index].Pos[0].Entr1_Ap_Pos[0] := "I_RPF_VASP_BR02";
	"DB_BIBLIOTHEQUE".Mobile[#index].Pos[0].Sort0[0] := "I_CO_VASP_BR02";
	"DB_BIBLIOTHEQUE".Mobile[#index].Pos[0].Sort0_Pr_Fin_Pos[0] := "I_CO_VASP_BR02";

	//position ouverture
	"DB_BIBLIOTHEQUE".Mobile[#index].Pos[1].Entr0_Ap_Pos[0] := "I_RPF_VASP_BR02";
	"DB_BIBLIOTHEQUE".Mobile[#index].Pos[1].Entr1_Ap_Pos[0] := "I_RPO_VASP_BR02";
	"DB_BIBLIOTHEQUE".Mobile[#index].Pos[1].Sort1[0] := "I_CO_VASP_BR02";
	"DB_BIBLIOTHEQUE".Mobile[#index].Pos[1].Sort0_Pr_Fin_Pos[0] := "I_CO_VASP_BR02";
	#index := #index + 1;
	//++++++++++++++++++++++++++++++++++++++++++++++++++++++++++++++/*296*/
	"DB_BIBLIOTHEQUE".Mobile[#index].Nom := 'VENT_BR2';
	"DB_BIBLIOTHEQUE".Mobile[#index].Pos[0].Nom := 'MARCHE';
	"DB_BIBLIOTHEQUE".Mobile[#index].Tjr_Desasservi := TRUE;
	"Init_Tps"(#index);

	// Entrées avant pos
	"DB_BIBLIOTHEQUE".Mobile[#index].Pos[0].Entr0_Av_Pos[0] := "I_RD_DISJ_VENT_BR02";

	// Entrées apres pos
	"DB_BIBLIOTHEQUE".Mobile[#index].Pos[0].Entr0_Ap_Pos[1] := "I_RD_DISJ_VENT_BR02";
	"DB_BIBLIOTHEQUE".Mobile[#index].Pos[0].Entr1_Ap_Pos[0] := "I_RM_VENT_BR02";

	// Entrées fin pos
	"DB_BIBLIOTHEQUE".Mobile[#index].Pos[0].Entr0_Ap_Fin_Pos[0] := "I_RM_VENT_BR02";

	// Sorties
	"DB_BIBLIOTHEQUE".Mobile[#index].Pos[0].Sort1[0] := "I_CM_VENT_BR02";
	"DB_BIBLIOTHEQUE".Mobile[#index].Pos[0].Sort0_Pr_Fin_Pos[0] := "I_CM_VENT_BR02";
	#index := #index + 1;
	//++++++++++++++++++++++++++++++++++++++++++++++++++++++++++++++/*297*/
	"DB_BIBLIOTHEQUE".Mobile[#index].Nom := 'DECOL_BR2';
	"DB_BIBLIOTHEQUE".Mobile[#index].Pos[0].Nom := 'MARCHE';
	"DB_BIBLIOTHEQUE".Mobile[#index].Tjr_Desasservi := TRUE;
	"Init_Tps"(#index);

	// Entrées fin pos
	"DB_BIBLIOTHEQUE".Mobile[#index].Pos[0].Entr0_Ap_Fin_Pos[0] := "I_RM_DECOL_BR02";

	// Sorties
	"DB_BIBLIOTHEQUE".Mobile[#index].Pos[0].Sort1[0] := "I_CM_DECOL_BR02";
	"DB_BIBLIOTHEQUE".Mobile[#index].Pos[0].Sort0_Pr_Fin_Pos[0] := "I_CM_DECOL_BR02";
	#index := #index + 1;
	//++++++++++++++++++++++++++++++++++++++++++++++++++++++++++++++/*298*/
	"DB_BIBLIOTHEQUE".Mobile[#index].Nom := 'VIB_BR2';
	"DB_BIBLIOTHEQUE".Mobile[#index].Pos[0].Nom := 'FERMETURE';
	"DB_BIBLIOTHEQUE".Mobile[#index].Pos[1].Nom := 'OUVERTURE';
	"DB_BIBLIOTHEQUE".Mobile[#index].Tjr_Desasservi := TRUE;
	"Init_Tps"(#index);
	#index := #index + 1;
	//++++++++++++++++++++++++++++++++++++++++++++++++++++++++++++++/*299*/
	"DB_BIBLIOTHEQUE".Mobile[#index].Nom := 'Vis_Ep_BR2';
	"DB_BIBLIOTHEQUE".Mobile[#index].Pos[0].Nom := 'MARCHE';
	"DB_BIBLIOTHEQUE".Mobile[#index].Tjr_Desasservi := TRUE;
	"Init_Tps"(#index);

	// Entrées avant pos
	"DB_BIBLIOTHEQUE".Mobile[#index].Pos[0].Entr0_Av_Pos[0] := "I_RD_DISJ_EPIER_BR02";

	// Entrées apres pos
	"DB_BIBLIOTHEQUE".Mobile[#index].Pos[0].Entr0_Ap_Pos[1] := "I_RD_DISJ_EPIER_BR02";
	// "DB_BIBLIOTHEQUE".Mobile[#index].Pos[0].Entr1_Ap_Pos[0] := "I_RR_EPIER_BR02";
	"DB_BIBLIOTHEQUE".Mobile[#index].Pos[0].Entr1_Ap_Pos[0] := "I_RM_EPIER_BR02";

	// Entrées fin pos
	"DB_BIBLIOTHEQUE".Mobile[#index].Pos[0].Entr0_Ap_Fin_Pos[0] := "I_RM_EPIER_BR02";

	// Sorties
	"DB_BIBLIOTHEQUE".Mobile[#index].Pos[0].Sort1[0] := "I_CM_EPIER_BR02";
	"DB_BIBLIOTHEQUE".Mobile[#index].Pos[0].Sort0_Pr_Fin_Pos[0] := "I_CM_EPIER_BR02";
	#index := #index + 1;
	//++++++++++++++++++++++++++++++++++++++++++++++++++++++++++++++/*300*/
	"DB_BIBLIOTHEQUE".Mobile[#index].Nom := 'MAGNET_BR2';
	// "DB_BIBLIOTHEQUE".Mobile[#index].Mob_Suiv[0] := "Index_Mobile"('TMEL');
	// "DB_BIBLIOTHEQUE".Mobile[#index].Pos[0].Nom := 'DROITE';
	// "DB_BIBLIOTHEQUE".Mobile[#index].Pos[0].Mob_Suiv[0] := "Index_Mobile"('TMEL');
	//"DB_BIBLIOTHEQUE".Mobile[#index].Tjr_Desasservi := TRUE;
	// "DB_BIBLIOTHEQUE".Mobile[#index].Tps_Att := t#500ms;
	// "DB_BIBLIOTHEQUE".Mobile[#index].Tps_Arr := t#0ms;

	// Entrées fin pos
	// "DB_BIBLIOTHEQUE".Mobile[#index].Pos[0].Entr0_Ap_Fin_Pos[0] := "I_RM_MAGN_BR02";

	// Sorties
	"DB_BIBLIOTHEQUE".Mobile[#index].Pos[0].Sort1[0] := "I_CM_MAGNET_BR02";
	"DB_BIBLIOTHEQUE".Mobile[#index].Pos[0].Sort0_Pr_Fin_Pos[0] := "I_CM_MAGNET_BR02";
	#index := #index + 1;

	//++++++++++++++++++++++++++++++++++++++++++++++++++++++++++++++/*301*/
	"DB_BIBLIOTHEQUE".Mobile[#index].Nom := 'T24';
	"DB_BIBLIOTHEQUE".Mobile[#index].Mob_Suiv[0] := "Index_Mobile"('E11');
	"DB_BIBLIOTHEQUE".Mobile[#index].Pos[0].Nom := 'DROITE';
	"DB_BIBLIOTHEQUE".Mobile[#index].Pos[0].Mob_Suiv[0] := "Index_Mobile"('E11');
	"DB_BIBLIOTHEQUE".Mobile[#index].Pos[0].Suiv_Enc := "Index_Mobile"('E11');
	// "DB_BIBLIOTHEQUE".Mobile[#index].Pass_Mat := "RPM_T24";
	"DB_BIBLIOTHEQUE".Mobile[#index].Tps_Att := t#5s;
	"DB_BIBLIOTHEQUE".Mobile[#index].Tps_Arr := t#0ms;

	// Entrées avant pos
	"DB_BIBLIOTHEQUE".Mobile[#index].Pos[0].Entr0_Av_Pos[0] := "I_RD_DISJ_T24";

	// Entrées apres pos
	"DB_BIBLIOTHEQUE".Mobile[#index].Pos[0].Entr0_Ap_Pos[0] := "I_RB_T24";
	"DB_BIBLIOTHEQUE".Mobile[#index].Pos[0].Entr0_Ap_Pos[1] := "I_RD_DISJ_T24";

	// "DB_BIBLIOTHEQUE".Mobile[#index].Pos[0].Entr1_Ap_Pos[0] := "I_RR_T24";
	"DB_BIBLIOTHEQUE".Mobile[#index].Pos[0].Entr1_Ap_Pos[0] := "I_RM_T24";

	// Entrées fin pos
	//"DB_BIBLIOTHEQUE".Mobile[#index].Pos[0].Entr0_Ap_Fin_Pos[0]:="I_RM_T24";

	// Sorties
	"DB_BIBLIOTHEQUE".Mobile[#index].Pos[0].Sort1[0] := "I_CM_T24";
	"DB_BIBLIOTHEQUE".Mobile[#index].Pos[0].Sort0_Pr_Fin_Pos[0] := "I_CM_T24";
	#index := #index + 1;
	//++++++++++++++++++++++++++++++++++++++++++++++++++++++++++++++/*302*/
	"DB_BIBLIOTHEQUE".Mobile[#index].Nom := 'T25';
	"DB_BIBLIOTHEQUE".Mobile[#index].Mob_Suiv[0] := "Index_Mobile"('E11');
	"DB_BIBLIOTHEQUE".Mobile[#index].Pos[0].Nom := 'DROIT';
	"DB_BIBLIOTHEQUE".Mobile[#index].Pos[0].Mob_Suiv[0] := "Index_Mobile"('E11');
	"DB_BIBLIOTHEQUE".Mobile[#index].Pos[0].Suiv_Enc := "Index_Mobile"('E11');
	"DB_BIBLIOTHEQUE".Mobile[#index].Tps_Att := t#500ms;
	"DB_BIBLIOTHEQUE".Mobile[#index].Tps_Arr := t#0ms;
	"DB_BIBLIOTHEQUE".Mobile[#index].Pass_Mat := "RPM_T25";

	// Entrées avant pos
	"DB_BIBLIOTHEQUE".Mobile[#index].Pos[0].Entr0_Av_Pos[0] := "I_RD_DISJ_T25";

	// Entrées apres pos
	"DB_BIBLIOTHEQUE".Mobile[#index].Pos[0].Entr0_Ap_Pos[0] := "I_RB_T25";
	"DB_BIBLIOTHEQUE".Mobile[#index].Pos[0].Entr0_Ap_Pos[1] := "I_RD_DISJ_T25";
	// "DB_BIBLIOTHEQUE".Mobile[#index].Pos[0].Entr1_Ap_Pos[0] := "I_RR_T25";
	"DB_BIBLIOTHEQUE".Mobile[#index].Pos[0].Entr1_Ap_Pos[0] := "I_RM_T25";

	// Entrées fin pos
	"DB_BIBLIOTHEQUE".Mobile[#index].Pos[0].Entr0_Ap_Fin_Pos[0] := "I_RM_T25";

	// Sorties
	"DB_BIBLIOTHEQUE".Mobile[#index].Pos[0].Sort1[0] := "I_CM_T25";
	"DB_BIBLIOTHEQUE".Mobile[#index].Pos[0].Sort0_Pr_Fin_Pos[0] := "I_CM_T25";
	#index := #index + 1;
	//++++++++++++++++++++++++++++++++++++++++++++++++++++++++++++++/*303*/
	"DB_BIBLIOTHEQUE".Mobile[#index].Nom := 'T27';
	"DB_BIBLIOTHEQUE".Mobile[#index].Mob_Suiv[0] := "Index_Mobile"('O_Exp_Fict');
	"DB_BIBLIOTHEQUE".Mobile[#index].Pos[0].Nom := 'MARCHE';
	"DB_BIBLIOTHEQUE".Mobile[#index].Pos[0].Mob_Suiv[0] := "Index_Mobile"('O_Exp_Fict');
	"DB_BIBLIOTHEQUE".Mobile[#index].Pos[0].Suiv_Enc := "Index_Mobile"('O_Exp_Fict');
	// "DB_BIBLIOTHEQUE".Mobile[#index].Pass_Mat := "RPM_T27";
	"DB_BIBLIOTHEQUE".Mobile[#index].Tps_Att := t#500ms;
	"DB_BIBLIOTHEQUE".Mobile[#index].Tps_Arr := t#0ms;

	// Entrées avant pos
	"DB_BIBLIOTHEQUE".Mobile[#index].Pos[0].Entr0_Av_Pos[0] := "I_RD_DISJ_T27";

	// Entrées apres pos
	"DB_BIBLIOTHEQUE".Mobile[#index].Pos[0].Entr0_Ap_Pos[0] := "I_RB_T27";
	"DB_BIBLIOTHEQUE".Mobile[#index].Pos[0].Entr0_Ap_Pos[1] := "I_RD_DISJ_T27";

	// "DB_BIBLIOTHEQUE".Mobile[#index].Pos[0].Entr1_Ap_Pos[0] := "I_RR_T27";
	"DB_BIBLIOTHEQUE".Mobile[#index].Pos[0].Entr1_Ap_Pos[0] := "I_RM_T27";

	// Entrées fin pos
	"DB_BIBLIOTHEQUE".Mobile[#index].Pos[0].Entr0_Ap_Fin_Pos[0] := "I_RM_T27";

	// Sorties
	"DB_BIBLIOTHEQUE".Mobile[#index].Pos[0].Sort1[0] := "I_CM_T27";
	"DB_BIBLIOTHEQUE".Mobile[#index].Pos[0].Sort0_Pr_Fin_Pos[0] := "I_CM_T27";
	#index := #index + 1;
	//++++++++++++++++++++++++++++++++++++++++++++++++++++++++++++++/*304*/
	"DB_BIBLIOTHEQUE".Mobile[#index].Nom := 'T28';
	"DB_BIBLIOTHEQUE".Mobile[#index].Noeud := TRUE;
	"DB_BIBLIOTHEQUE".Mobile[#index].Mob_Suiv[0] := "Index_Mobile"('TRP1_T28');
	"DB_BIBLIOTHEQUE".Mobile[#index].Mob_Suiv[1] := "Index_Mobile"('TRP2_T28');
	"DB_BIBLIOTHEQUE".Mobile[#index].Mob_Suiv[2] := "Index_Mobile"('TRP3_T28');
	"DB_BIBLIOTHEQUE".Mobile[#index].Mob_Suiv[3] := "Index_Mobile"('TRP4_T28');
	"DB_BIBLIOTHEQUE".Mobile[#index].Mob_Suiv[4] := "Index_Mobile"('TRP5_T28');
	"DB_BIBLIOTHEQUE".Mobile[#index].Pos[0].Nom := 'DROITE';
	"DB_BIBLIOTHEQUE".Mobile[#index].Pos[0].Mob_Suiv[0] := "Index_Mobile"('TRP1_T28');
	"DB_BIBLIOTHEQUE".Mobile[#index].Pos[0].Mob_Suiv[1] := "Index_Mobile"('TRP2_T28');
	"DB_BIBLIOTHEQUE".Mobile[#index].Pos[0].Mob_Suiv[2] := "Index_Mobile"('TRP3_T28');
	"DB_BIBLIOTHEQUE".Mobile[#index].Pos[0].Mob_Suiv[3] := "Index_Mobile"('TRP4_T28');
	"DB_BIBLIOTHEQUE".Mobile[#index].Pos[0].Mob_Suiv[4] := "Index_Mobile"('TRP5_T28');


	// Entrées avant pos
	"DB_BIBLIOTHEQUE".Mobile[#index].Pos[0].Entr0_Av_Pos[0] := "I_RD_DISJ_T28";

	// Entrées apres pos
	"DB_BIBLIOTHEQUE".Mobile[#index].Pos[0].Entr0_Ap_Pos[0] := "I_RB_T28";
	"DB_BIBLIOTHEQUE".Mobile[#index].Pos[0].Entr0_Ap_Pos[1] := "I_RD_DISJ_T28";

	// "DB_BIBLIOTHEQUE".Mobile[#index].Pos[0].Entr1_Ap_Pos[0] := "I_RR_T28";
	"DB_BIBLIOTHEQUE".Mobile[#index].Pos[0].Entr1_Ap_Pos[0] := "I_RM_T28";

	// Entrées fin pos
	"DB_BIBLIOTHEQUE".Mobile[#index].Pos[0].Entr0_Ap_Fin_Pos[0] := "I_RM_T28";

	// Sorties
	"DB_BIBLIOTHEQUE".Mobile[#index].Pos[0].Sort1[0] := "I_CM_T28";
	"DB_BIBLIOTHEQUE".Mobile[#index].Pos[0].Sort0_Pr_Fin_Pos[0] := "I_CM_T28";
	#index := #index + 1;
	//++++++++++++++++++++++++++++++++++++++++++++++++++++++++++++++/*305*/
	"DB_BIBLIOTHEQUE".Mobile[#index].Nom := 'T29';
	"DB_BIBLIOTHEQUE".Mobile[#index].Noeud := TRUE;
	"DB_BIBLIOTHEQUE".Mobile[#index].Mob_Suiv[0] := "Index_Mobile"('TRP1_T29');
	"DB_BIBLIOTHEQUE".Mobile[#index].Mob_Suiv[1] := "Index_Mobile"('TRP2_T29');
	"DB_BIBLIOTHEQUE".Mobile[#index].Pos[0].Nom := 'DROIT';
	"DB_BIBLIOTHEQUE".Mobile[#index].Pos[0].Mob_Suiv[0] := "Index_Mobile"('TRP1_T29');
	"DB_BIBLIOTHEQUE".Mobile[#index].Pos[0].Mob_Suiv[1] := "Index_Mobile"('TRP2_T29');
	"Init_Tps"(#index);

	// Entrées avant pos
	"DB_BIBLIOTHEQUE".Mobile[#index].Pos[0].Entr0_Av_Pos[0] := "I_RD_DISJ_T29";
	"DB_BIBLIOTHEQUE".Mobile[#index].Pos[0].Entr0_Av_Pos[1] := "I_RD_DISJ_T29";
	// Entrées apres pos
	"DB_BIBLIOTHEQUE".Mobile[#index].Pos[0].Entr0_Ap_Pos[0] := "I_RB_T29";
	"DB_BIBLIOTHEQUE".Mobile[#index].Pos[0].Entr0_Ap_Pos[1] := "I_RD_DISJ_T29";
	// "DB_BIBLIOTHEQUE".Mobile[#index].Pos[0].Entr1_Ap_Pos[0] := "I_RR_T29";
	"DB_BIBLIOTHEQUE".Mobile[#index].Pos[0].Entr1_Ap_Pos[0] := "I_RM_T29";
	// Entrées fin pos
	"DB_BIBLIOTHEQUE".Mobile[#index].Pos[0].Entr0_Ap_Fin_Pos[0] := "I_RM_T29";
	// Sorties
	"DB_BIBLIOTHEQUE".Mobile[#index].Pos[0].Sort1[0] := "I_CM_T29";
	"DB_BIBLIOTHEQUE".Mobile[#index].Pos[0].Sort0_Pr_Fin_Pos[0] := "I_CM_T29";
	#index := #index + 1;
	//++++++++++++++++++++++++++++++++++++++++++++++++++++++++++++++/*306*/
	"DB_BIBLIOTHEQUE".Mobile[#index].Nom := 'T42';
	"DB_BIBLIOTHEQUE".Mobile[#index].Noeud := TRUE;
	"DB_BIBLIOTHEQUE".Mobile[#index].Mob_Suiv[0] := "Index_Mobile"('TRP1_T42');
	"DB_BIBLIOTHEQUE".Mobile[#index].Mob_Suiv[1] := "Index_Mobile"('TRP2_T42');
	"DB_BIBLIOTHEQUE".Mobile[#index].Mob_Suiv[2] := "Index_Mobile"('TRP3_T42');
	"DB_BIBLIOTHEQUE".Mobile[#index].Pos[0].Nom := 'DROIT';
	"DB_BIBLIOTHEQUE".Mobile[#index].Pos[0].Mob_Suiv[0] := "Index_Mobile"('TRP1_T42');
	"DB_BIBLIOTHEQUE".Mobile[#index].Pos[0].Mob_Suiv[1] := "Index_Mobile"('TRP2_T42');
	"DB_BIBLIOTHEQUE".Mobile[#index].Pos[0].Mob_Suiv[2] := "Index_Mobile"('TRP3_T42');
	"DB_BIBLIOTHEQUE".Mobile[#index].Tps_Att := t#500ms;
	"DB_BIBLIOTHEQUE".Mobile[#index].Tps_Arr := t#0ms;

	// Entrées avant pos
	"DB_BIBLIOTHEQUE".Mobile[#index].Pos[0].Entr0_Av_Pos[0] := "I_RD_DISJ_T42";
	// Entrées apres pos
	"DB_BIBLIOTHEQUE".Mobile[#index].Pos[0].Entr0_Ap_Pos[0] := "I_RB_T42";
	"DB_BIBLIOTHEQUE".Mobile[#index].Pos[0].Entr0_Ap_Pos[1] := "I_RD_DISJ_T42";
	// "DB_BIBLIOTHEQUE".Mobile[#index].Pos[0].Entr1_Ap_Pos[0] := "I_RR_T42";
	"DB_BIBLIOTHEQUE".Mobile[#index].Pos[0].Entr1_Ap_Pos[0] := "I_RM_T42";
	// Entrées fin pos
	"DB_BIBLIOTHEQUE".Mobile[#index].Pos[0].Entr0_Ap_Fin_Pos[0] := "I_RM_T42";
	// Sorties
	"DB_BIBLIOTHEQUE".Mobile[#index].Pos[0].Sort1[0] := "I_CM_T42";
	"DB_BIBLIOTHEQUE".Mobile[#index].Pos[0].Sort0_Pr_Fin_Pos[0] := "I_CM_T42";
	#index := #index + 1;
	//++++++++++++++++++++++++++++++++++++++++++++++++++++++++++++++/*307*/
	"DB_BIBLIOTHEQUE".Mobile[#index].Nom := 'T48';
	"DB_BIBLIOTHEQUE".Mobile[#index].Mob_Suiv[0] := "Index_Mobile"('E24');
	"DB_BIBLIOTHEQUE".Mobile[#index].Pos[0].Nom := 'DROIT';
	"DB_BIBLIOTHEQUE".Mobile[#index].Pos[0].Mob_Suiv[0] := "Index_Mobile"('E24');
	"Init_Tps"(#index);

	// Entrées avant pos
	"DB_BIBLIOTHEQUE".Mobile[#index].Pos[0].Entr0_Av_Pos[0] := "I_RD_DISJ_T48";
	// Entrées apres pos
	// "DB_BIBLIOTHEQUE".Mobile[#index].Pos[0].Entr0_Ap_Pos[0] := "I_RB_T48";
	"DB_BIBLIOTHEQUE".Mobile[#index].Pos[0].Entr0_Ap_Pos[1] := "I_RD_DISJ_T48";
	// "DB_BIBLIOTHEQUE".Mobile[#index].Pos[0].Entr1_Ap_Pos[0] := "I_RR_T48";
	"DB_BIBLIOTHEQUE".Mobile[#index].Pos[0].Entr1_Ap_Pos[0] := "I_RM_T48";
	// Entrées fin pos
	"DB_BIBLIOTHEQUE".Mobile[#index].Pos[0].Entr0_Ap_Fin_Pos[0] := "I_RM_T48";
	// Sorties
	"DB_BIBLIOTHEQUE".Mobile[#index].Pos[0].Sort1[0] := "I_CM_T48";
	"DB_BIBLIOTHEQUE".Mobile[#index].Pos[0].Sort0_Pr_Fin_Pos[0] := "I_CM_T48";
	#index := #index + 1;
	//++++++++++++++++++++++++++++++++++++++++++++++++++++++++++++++/*308*/
	"DB_BIBLIOTHEQUE".Mobile[#index].Nom := 'E12';
	"DB_BIBLIOTHEQUE".Mobile[#index].Mob_Suiv[0] := "Index_Mobile"('T28');
	"DB_BIBLIOTHEQUE".Mobile[#index].Pos[0].Nom := 'MARCHE';
	"DB_BIBLIOTHEQUE".Mobile[#index].Pos[0].Mob_Suiv[0] := "Index_Mobile"('T28');

	// Entrées avant pos
	"DB_BIBLIOTHEQUE".Mobile[#index].Pos[0].Entr0_Av_Pos[0] := "I_RD_DISJ_E12";
	"DB_BIBLIOTHEQUE".Mobile[#index].Pos[0].Entr0_Av_Pos[1] := "I_RD_DBHG_E12";
	"DB_BIBLIOTHEQUE".Mobile[#index].Pos[0].Entr0_Av_Pos[2] := "I_RD_DBHD_E12";
	"DB_BIBLIOTHEQUE".Mobile[#index].Pos[0].Entr0_Av_Pos[3] := "I_RD_DBBG_E12";
	"DB_BIBLIOTHEQUE".Mobile[#index].Pos[0].Entr0_Av_Pos[4] := "I_RD_DBBD_E12";

	// Entrées apres pos
	"DB_BIBLIOTHEQUE".Mobile[#index].Pos[0].Entr0_Ap_Pos[0] := "I_RD_DISJ_E12";
	"DB_BIBLIOTHEQUE".Mobile[#index].Pos[0].Entr0_Ap_Pos[1] := "I_RD_DBHG_E12";
	"DB_BIBLIOTHEQUE".Mobile[#index].Pos[0].Entr0_Ap_Pos[2] := "I_RD_DBHD_E12";
	"DB_BIBLIOTHEQUE".Mobile[#index].Pos[0].Entr0_Ap_Pos[3] := "I_RD_DBBG_E12";
	"DB_BIBLIOTHEQUE".Mobile[#index].Pos[0].Entr0_Ap_Pos[4] := "I_RD_DBBD_E12";
	"DB_BIBLIOTHEQUE".Mobile[#index].Pos[0].Entr1_Ap_Pos[0] := "I_RR_E12";
	"DB_BIBLIOTHEQUE".Mobile[#index].Pos[0].Entr1_Ap_Pos[1] := "I_RM_E12";

	// Entrées fin pos
	"DB_BIBLIOTHEQUE".Mobile[#index].Pos[0].Entr0_Ap_Fin_Pos[0] := "I_RM_E12";

	// Sorties
	"DB_BIBLIOTHEQUE".Mobile[#index].Pos[0].Sort1[0] := "I_CM_E12";
	"DB_BIBLIOTHEQUE".Mobile[#index].Pos[0].Sort0_Pr_Fin_Pos[0] := "I_CM_E12";
	#index := #index + 1;
	//++++++++++++++++++++++++++++++++++++++++++++++++++++++++++++++/*309*/
	"DB_BIBLIOTHEQUE".Mobile[#index].Nom := 'TRP1_BP4';
	"DB_BIBLIOTHEQUE".Mobile[#index].Pos[0].Nom := 'FERMETURE';
	"DB_BIBLIOTHEQUE".Mobile[#index].Pos[1].Nom := 'OUVERTURE';
	"DB_BIBLIOTHEQUE".Mobile[#index].Tjr_Desasservi := TRUE;
	"Init_Tps"(#index);

	//position fermeture
	"DB_BIBLIOTHEQUE".Mobile[#index].Pos[0].Entr0_Ap_Pos[0] := "I_RPO_TRBP4";
	"DB_BIBLIOTHEQUE".Mobile[#index].Pos[0].Entr1_Ap_Pos[0] := "I_RPF_TRBP4";
	"DB_BIBLIOTHEQUE".Mobile[#index].Pos[0].Sort0[0] := "I_CO_TRBP4";
	"DB_BIBLIOTHEQUE".Mobile[#index].Pos[0].Sort0_Pr_Fin_Pos[0] := "I_CO_TRBP4";

	//position ouverture
	"DB_BIBLIOTHEQUE".Mobile[#index].Pos[1].Entr0_Ap_Pos[0] := "I_RPF_TRBP4";
	"DB_BIBLIOTHEQUE".Mobile[#index].Pos[1].Entr1_Ap_Pos[0] := "I_RPO_TRBP4";
	"DB_BIBLIOTHEQUE".Mobile[#index].Pos[1].Sort1[0] := "I_CO_TRBP4";
	"DB_BIBLIOTHEQUE".Mobile[#index].Pos[1].Sort0_Pr_Fin_Pos[0] := "I_CO_TRBP4";
	#index := #index + 1;
	//++++++++++++++++++++++++++++++++++++++++++++++++++++++++++++++/*310*/
	"DB_BIBLIOTHEQUE".Mobile[#index].Nom := 'TRP1_TBP4';
	"DB_BIBLIOTHEQUE".Mobile[#index].Pos[0].Nom := 'FERMETURE';
	"DB_BIBLIOTHEQUE".Mobile[#index].Pos[1].Nom := 'OUVERTURE';
	"DB_BIBLIOTHEQUE".Mobile[#index].Tjr_Desasservi := TRUE;
	"Init_Tps"(#index);

	//position fermeture
	"DB_BIBLIOTHEQUE".Mobile[#index].Pos[0].Entr0_Ap_Pos[0] := "I_RPO_TR_TRMBP4";
	"DB_BIBLIOTHEQUE".Mobile[#index].Pos[0].Entr1_Ap_Pos[0] := "I_RPF_TR_TRMBP4";
	"DB_BIBLIOTHEQUE".Mobile[#index].Pos[0].Sort0[0] := "I_CO_TR_TRMBP4";
	"DB_BIBLIOTHEQUE".Mobile[#index].Pos[0].Sort0_Pr_Fin_Pos[0] := "I_CO_TR_TRMBP4";

	//position ouverture
	"DB_BIBLIOTHEQUE".Mobile[#index].Pos[1].Entr0_Ap_Pos[0] := "I_RPF_TR_TRMBP4";
	"DB_BIBLIOTHEQUE".Mobile[#index].Pos[1].Entr1_Ap_Pos[0] := "I_RPO_TR_TRMBP4";
	"DB_BIBLIOTHEQUE".Mobile[#index].Pos[1].Sort1[0] := "I_CO_TR_TRMBP4";
	"DB_BIBLIOTHEQUE".Mobile[#index].Pos[1].Sort0_Pr_Fin_Pos[0] := "I_CO_TR_TRMBP4";
	#index := #index + 1;
	//++++++++++++++++++++++++++++++++++++++++++++++++++++++++++++++/*311*/
	"DB_BIBLIOTHEQUE".Mobile[#index].Nom := 'TRP1_T28';
	"DB_BIBLIOTHEQUE".Mobile[#index].Mob_Suiv[0] := "Index_Mobile"('BP01');
	"DB_BIBLIOTHEQUE".Mobile[#index].Pos[0].Nom := 'FERMETURE';
	"DB_BIBLIOTHEQUE".Mobile[#index].Pos[0].Mob_Suiv[0] := "Index_Mobile"('BP01');
	"DB_BIBLIOTHEQUE".Mobile[#index].Pos[1].Nom := 'OUVERTURE';
	"DB_BIBLIOTHEQUE".Mobile[#index].Pos[1].Mob_Suiv[0] := "Index_Mobile"('BP01');
	"Init_Tps"(#index);

	//position fermeture
	"DB_BIBLIOTHEQUE".Mobile[#index].Pos[0].Entr0_Ap_Pos[0] := "I_RPO_TRP1T28";
	"DB_BIBLIOTHEQUE".Mobile[#index].Pos[0].Entr1_Ap_Pos[0] := "I_RPF_TRP1T28";
	"DB_BIBLIOTHEQUE".Mobile[#index].Pos[0].Sort0[0] := "I_CO_TRP1T28";
	"DB_BIBLIOTHEQUE".Mobile[#index].Pos[0].Sort0_Pr_Fin_Pos[0] := "I_CO_TRP1T28";

	//position ouverture
	"DB_BIBLIOTHEQUE".Mobile[#index].Pos[1].Entr0_Ap_Pos[0] := "I_RPF_TRP1T28";
	"DB_BIBLIOTHEQUE".Mobile[#index].Pos[1].Entr1_Ap_Pos[0] := "I_RPO_TRP1T28";
	"DB_BIBLIOTHEQUE".Mobile[#index].Pos[1].Sort1[0] := "I_CO_TRP1T28";
	"DB_BIBLIOTHEQUE".Mobile[#index].Pos[1].Sort0_Pr_Fin_Pos[0] := "I_CO_TRP1T28";
	#index := #index + 1;
	//++++++++++++++++++++++++++++++++++++++++++++++++++++++++++++++/*312*/
	"DB_BIBLIOTHEQUE".Mobile[#index].Nom := 'TRP2_T28';
	"DB_BIBLIOTHEQUE".Mobile[#index].Mob_Suiv[0] := "Index_Mobile"('BP02');
	"DB_BIBLIOTHEQUE".Mobile[#index].Pos[0].Nom := 'FERMETURE';
	"DB_BIBLIOTHEQUE".Mobile[#index].Pos[0].Mob_Suiv[0] := "Index_Mobile"('BP02');
	"DB_BIBLIOTHEQUE".Mobile[#index].Pos[1].Nom := 'OUVERTURE';
	"DB_BIBLIOTHEQUE".Mobile[#index].Pos[1].Mob_Suiv[0] := "Index_Mobile"('BP02');
	"Init_Tps"(#index);

	//position fermeture
	"DB_BIBLIOTHEQUE".Mobile[#index].Pos[0].Entr0_Ap_Pos[0] := "I_RPO_TRP2T28";
	"DB_BIBLIOTHEQUE".Mobile[#index].Pos[0].Entr1_Ap_Pos[0] := "I_RPF_TRP2T28";
	"DB_BIBLIOTHEQUE".Mobile[#index].Pos[0].Sort0[0] := "I_CO_TRP2T28";
	"DB_BIBLIOTHEQUE".Mobile[#index].Pos[0].Sort0_Pr_Fin_Pos[0] := "I_CO_TRP2T28";

	//position ouverture
	"DB_BIBLIOTHEQUE".Mobile[#index].Pos[1].Entr0_Ap_Pos[0] := "I_RPF_TRP2T28";
	"DB_BIBLIOTHEQUE".Mobile[#index].Pos[1].Entr1_Ap_Pos[0] := "I_RPO_TRP2T28";
	"DB_BIBLIOTHEQUE".Mobile[#index].Pos[1].Sort1[0] := "I_CO_TRP2T28";
	"DB_BIBLIOTHEQUE".Mobile[#index].Pos[1].Sort0_Pr_Fin_Pos[0] := "I_CO_TRP2T28";
	#index := #index + 1;
	//++++++++++++++++++++++++++++++++++++++++++++++++++++++++++++++/*313*/
	"DB_BIBLIOTHEQUE".Mobile[#index].Nom := 'TRP3_T28';
	"DB_BIBLIOTHEQUE".Mobile[#index].Mob_Suiv[0] := "Index_Mobile"('T42');
	"DB_BIBLIOTHEQUE".Mobile[#index].Pos[0].Nom := 'FERMETURE';
	"DB_BIBLIOTHEQUE".Mobile[#index].Pos[1].Nom := 'OUVERTURE';
	"DB_BIBLIOTHEQUE".Mobile[#index].Pos[1].Mob_Suiv[0] := "Index_Mobile"('T42');
	"Init_Tps"(#index);
	"DB_BIBLIOTHEQUE".Mobile[#index].Tps_Vid := t#1s;

	//position fermeture
	"DB_BIBLIOTHEQUE".Mobile[#index].Pos[0].Entr0_Ap_Pos[0] := "I_RPO_TRP3T28";
	"DB_BIBLIOTHEQUE".Mobile[#index].Pos[0].Entr1_Ap_Pos[0] := "I_RPF_TRP3T28";
	"DB_BIBLIOTHEQUE".Mobile[#index].Pos[0].Sort0[0] := "I_CO_TRP3T28";
	"DB_BIBLIOTHEQUE".Mobile[#index].Pos[0].Sort0_Pr_Fin_Pos[0] := "I_CO_TRP3T28";

	//position ouverture
	"DB_BIBLIOTHEQUE".Mobile[#index].Pos[1].Entr0_Ap_Pos[0] := "I_RPF_TRP3T28";
	"DB_BIBLIOTHEQUE".Mobile[#index].Pos[1].Entr1_Ap_Pos[0] := "I_RPO_TRP3T28";
	"DB_BIBLIOTHEQUE".Mobile[#index].Pos[1].Sort1[0] := "I_CO_TRP3T28";
	"DB_BIBLIOTHEQUE".Mobile[#index].Pos[1].Sort0_Pr_Fin_Pos[0] := "I_CO_TRP3T28";
	#index := #index + 1;
	//++++++++++++++++++++++++++++++++++++++++++++++++++++++++++++++/*314*/
	"DB_BIBLIOTHEQUE".Mobile[#index].Nom := 'TRP4_T28';
	"DB_BIBLIOTHEQUE".Mobile[#index].Mob_Suiv[0] := "Index_Mobile"('T29');
	"DB_BIBLIOTHEQUE".Mobile[#index].Pos[0].Nom := 'FERMETURE';
	"DB_BIBLIOTHEQUE".Mobile[#index].Pos[0].Mob_Suiv[0] := "Index_Mobile"('T29');
	"DB_BIBLIOTHEQUE".Mobile[#index].Pos[1].Nom := 'OUVERTURE';
	"DB_BIBLIOTHEQUE".Mobile[#index].Pos[1].Mob_Suiv[0] := "Index_Mobile"('T29');
	"Init_Tps"(#index);

	//position fermeture
	"DB_BIBLIOTHEQUE".Mobile[#index].Pos[0].Entr0_Ap_Pos[0] := "I_RPO_TRP4T28";
	"DB_BIBLIOTHEQUE".Mobile[#index].Pos[0].Entr1_Ap_Pos[0] := "I_RPF_TRP4T28";
	"DB_BIBLIOTHEQUE".Mobile[#index].Pos[0].Sort0[0] := "I_CO_TRP4T28";
	"DB_BIBLIOTHEQUE".Mobile[#index].Pos[0].Sort0_Pr_Fin_Pos[0] := "I_CO_TRP4T28";

	//position ouverture
	"DB_BIBLIOTHEQUE".Mobile[#index].Pos[1].Entr0_Ap_Pos[0] := "I_RPF_TRP4T28";
	"DB_BIBLIOTHEQUE".Mobile[#index].Pos[1].Entr1_Ap_Pos[0] := "I_RPO_TRP4T28";
	"DB_BIBLIOTHEQUE".Mobile[#index].Pos[1].Sort1[0] := "I_CO_TRP4T28";
	"DB_BIBLIOTHEQUE".Mobile[#index].Pos[1].Sort0_Pr_Fin_Pos[0] := "I_CO_TRP4T28";
	#index := #index + 1;
	//++++++++++++++++++++++++++++++++++++++++++++++++++++++++++++++/*315*/
	"DB_BIBLIOTHEQUE".Mobile[#index].Nom := 'TRP5_T28';


	// //position fermeture
	// "DB_BIBLIOTHEQUE".Mobile[#index].Pos[0].Entr0_Ap_Pos[0] := "I_RPO_TRP5T28";
	// "DB_BIBLIOTHEQUE".Mobile[#index].Pos[0].Entr1_Ap_Pos[0] := "I_RPF_TRP5T28";
	// "DB_BIBLIOTHEQUE".Mobile[#index].Pos[0].Sort0[0] := "I_CO_TRP5T28";
	// "DB_BIBLIOTHEQUE".Mobile[#index].Pos[0].Sort0_Pr_Fin_Pos[0] := "I_CO_TRP5T28";

	// //position ouverture
	// "DB_BIBLIOTHEQUE".Mobile[#index].Pos[1].Entr0_Ap_Pos[0] := "I_RPF_TRP5T28";
	// "DB_BIBLIOTHEQUE".Mobile[#index].Pos[1].Entr1_Ap_Pos[0] := "I_RPO_TRP5T28";
	// "DB_BIBLIOTHEQUE".Mobile[#index].Pos[1].Sort1[0] := "I_CO_TRP5T28";
	// "DB_BIBLIOTHEQUE".Mobile[#index].Pos[1].Sort0_Pr_Fin_Pos[0] := "I_CO_TRP5T28";
	#index := #index + 1;
	//++++++++++++++++++++++++++++++++++++++++++++++++++++++++++++++/*316*/
	"DB_BIBLIOTHEQUE".Mobile[#index].Nom := 'TRP1_T42';
	"DB_BIBLIOTHEQUE".Mobile[#index].Mob_Suiv[0] := "Index_Mobile"('BT01');
	"DB_BIBLIOTHEQUE".Mobile[#index].Pos[0].Nom := 'FERMETURE';
	"DB_BIBLIOTHEQUE".Mobile[#index].Pos[1].Nom := 'OUVERTURE';
	"DB_BIBLIOTHEQUE".Mobile[#index].Pos[1].Mob_Suiv[0] := "Index_Mobile"('BT01');
	"Init_Tps"(#index);

	//position fermeture
	"DB_BIBLIOTHEQUE".Mobile[#index].Pos[0].Entr0_Ap_Pos[0] := "I_RPO_TRP1T42";
	"DB_BIBLIOTHEQUE".Mobile[#index].Pos[0].Entr1_Ap_Pos[0] := "I_RPF_TRP1T42";
	"DB_BIBLIOTHEQUE".Mobile[#index].Pos[0].Sort0[0] := "I_CO_TRP1T42";
	"DB_BIBLIOTHEQUE".Mobile[#index].Pos[0].Sort0_Pr_Fin_Pos[0] := "I_CO_TRP1T42";

	//position ouverture
	"DB_BIBLIOTHEQUE".Mobile[#index].Pos[1].Entr0_Ap_Pos[0] := "I_RPF_TRP1T42";
	"DB_BIBLIOTHEQUE".Mobile[#index].Pos[1].Entr1_Ap_Pos[0] := "I_RPO_TRP1T42";
	"DB_BIBLIOTHEQUE".Mobile[#index].Pos[1].Sort1[0] := "I_CO_TRP1T42";
	"DB_BIBLIOTHEQUE".Mobile[#index].Pos[1].Sort0_Pr_Fin_Pos[0] := "I_CO_TRP1T42";
	#index := #index + 1;
	//++++++++++++++++++++++++++++++++++++++++++++++++++++++++++++++/*317*/
	"DB_BIBLIOTHEQUE".Mobile[#index].Nom := 'TRP2_T42';
	"DB_BIBLIOTHEQUE".Mobile[#index].Mob_Suiv[0] := "Index_Mobile"('BT04');
	"DB_BIBLIOTHEQUE".Mobile[#index].Pos[0].Nom := 'FERMETURE';
	"DB_BIBLIOTHEQUE".Mobile[#index].Pos[1].Nom := 'OUVERTURE';
	"DB_BIBLIOTHEQUE".Mobile[#index].Pos[1].Mob_Suiv[0] := "Index_Mobile"('BT04');
	"Init_Tps"(#index);


	//position fermeture
	"DB_BIBLIOTHEQUE".Mobile[#index].Pos[0].Entr0_Ap_Pos[0] := "I_RPO_TRP2T42";
	"DB_BIBLIOTHEQUE".Mobile[#index].Pos[0].Entr1_Ap_Pos[0] := "I_RPF_TRP2T42";
	"DB_BIBLIOTHEQUE".Mobile[#index].Pos[0].Sort0[0] := "I_CO_TRP2T42";
	"DB_BIBLIOTHEQUE".Mobile[#index].Pos[0].Sort0_Pr_Fin_Pos[0] := "I_CO_TRP2T42";

	//position ouverture
	"DB_BIBLIOTHEQUE".Mobile[#index].Pos[1].Entr0_Ap_Pos[0] := "I_RPF_TRP2T42";
	"DB_BIBLIOTHEQUE".Mobile[#index].Pos[1].Entr1_Ap_Pos[0] := "I_RPO_TRP2T42";
	"DB_BIBLIOTHEQUE".Mobile[#index].Pos[1].Sort1[0] := "I_CO_TRP2T42";
	"DB_BIBLIOTHEQUE".Mobile[#index].Pos[1].Sort0_Pr_Fin_Pos[0] := "I_CO_TRP2T42";
	#index := #index + 1;
	//++++++++++++++++++++++++++++++++++++++++++++++++++++++++++++++/*318*/
	"DB_BIBLIOTHEQUE".Mobile[#index].Nom := 'TRP3_T42';
	"DB_BIBLIOTHEQUE".Mobile[#index].Mob_Suiv[0] := "Index_Mobile"('T48');
	"DB_BIBLIOTHEQUE".Mobile[#index].Pos[0].Nom := 'FERMETURE';
	"DB_BIBLIOTHEQUE".Mobile[#index].Pos[0].Mob_Suiv[0] := "Index_Mobile"('T48');
	"DB_BIBLIOTHEQUE".Mobile[#index].Pos[1].Nom := 'OUVERTURE';
	"DB_BIBLIOTHEQUE".Mobile[#index].Pos[1].Mob_Suiv[0] := "Index_Mobile"('T48');
	"Init_Tps"(#index);


	//position fermeture
	"DB_BIBLIOTHEQUE".Mobile[#index].Pos[0].Entr0_Ap_Pos[0] := "I_RPO_TRP3T42";
	"DB_BIBLIOTHEQUE".Mobile[#index].Pos[0].Entr1_Ap_Pos[0] := "I_RPF_TRP3T42";
	"DB_BIBLIOTHEQUE".Mobile[#index].Pos[0].Sort0[0] := "I_CO_TRP3T42";
	"DB_BIBLIOTHEQUE".Mobile[#index].Pos[0].Sort0_Pr_Fin_Pos[0] := "I_CO_TRP3T42";

	//position ouverture
	"DB_BIBLIOTHEQUE".Mobile[#index].Pos[1].Entr0_Ap_Pos[0] := "I_RPF_TRP3T42";
	"DB_BIBLIOTHEQUE".Mobile[#index].Pos[1].Entr1_Ap_Pos[0] := "I_RPO_TRP3T42";
	"DB_BIBLIOTHEQUE".Mobile[#index].Pos[1].Sort1[0] := "I_CO_TRP3T42";
	"DB_BIBLIOTHEQUE".Mobile[#index].Pos[1].Sort0_Pr_Fin_Pos[0] := "I_CO_TRP3T42";
	#index := #index + 1;
	//++++++++++++++++++++++++++++++++++++++++++++++++++++++++++++++/*319*/
	"DB_BIBLIOTHEQUE".Mobile[#index].Nom := 'TRP1_T29';
	"DB_BIBLIOTHEQUE".Mobile[#index].Mob_Suiv[0] := "Index_Mobile"('REV01');
	"DB_BIBLIOTHEQUE".Mobile[#index].Pos[0].Nom := 'FERMETURE';
	"DB_BIBLIOTHEQUE".Mobile[#index].Pos[0].Mob_Suiv[0] := "Index_Mobile"('REV01');
	"DB_BIBLIOTHEQUE".Mobile[#index].Pos[1].Nom := 'OUVERTURE';
	"DB_BIBLIOTHEQUE".Mobile[#index].Pos[1].Mob_Suiv[0] := "Index_Mobile"('REV01');
	"Init_Tps"(#index);


	//position fermeture
	"DB_BIBLIOTHEQUE".Mobile[#index].Pos[0].Entr0_Ap_Pos[0] := "I_RPO_TRP1T29";
	"DB_BIBLIOTHEQUE".Mobile[#index].Pos[0].Entr1_Ap_Pos[0] := "I_RPF_TRP1T29";
	"DB_BIBLIOTHEQUE".Mobile[#index].Pos[0].Sort0[0] := "I_CO_TRP1T29";
	"DB_BIBLIOTHEQUE".Mobile[#index].Pos[0].Sort0_Pr_Fin_Pos[0] := "I_CO_TRP1T29";

	//position ouverture
	"DB_BIBLIOTHEQUE".Mobile[#index].Pos[1].Entr0_Ap_Pos[0] := "I_RPF_TRP1T29";
	"DB_BIBLIOTHEQUE".Mobile[#index].Pos[1].Entr1_Ap_Pos[0] := "I_RPO_TRP1T29";
	"DB_BIBLIOTHEQUE".Mobile[#index].Pos[1].Sort1[0] := "I_CO_TRP1T29";
	"DB_BIBLIOTHEQUE".Mobile[#index].Pos[1].Sort0_Pr_Fin_Pos[0] := "I_CO_TRP1T29";
	#index := #index + 1;
	//++++++++++++++++++++++++++++++++++++++++++++++++++++++++++++++/*320*/
	"DB_BIBLIOTHEQUE".Mobile[#index].Nom := 'REV01';
	"DB_BIBLIOTHEQUE".Mobile[#index].Noeud := TRUE;//NOEUD
	"DB_BIBLIOTHEQUE".Mobile[#index].Mob_Suiv[0] := "Index_Mobile"('BT10');
	"DB_BIBLIOTHEQUE".Mobile[#index].Mob_Suiv[1] := "Index_Mobile"('BT17');
	"DB_BIBLIOTHEQUE".Mobile[#index].Mob_Suiv[2] := "Index_Mobile"('BT16');
	"DB_BIBLIOTHEQUE".Mobile[#index].Mob_Suiv[3] := "Index_Mobile"('BT12');

	"DB_BIBLIOTHEQUE".Mobile[#index].Pos[0].Nom := 'BT10';
	"DB_BIBLIOTHEQUE".Mobile[#index].Pos[0].Mob_Suiv[0] := "Index_Mobile"('BT10');
	"DB_BIBLIOTHEQUE".Mobile[#index].Pos[1].Nom := 'BT17';
	"DB_BIBLIOTHEQUE".Mobile[#index].Pos[1].Mob_Suiv[0] := "Index_Mobile"('BT17');
	"DB_BIBLIOTHEQUE".Mobile[#index].Pos[2].Nom := 'BT16';
	"DB_BIBLIOTHEQUE".Mobile[#index].Pos[2].Mob_Suiv[0] := "Index_Mobile"('BT16');
	"DB_BIBLIOTHEQUE".Mobile[#index].Pos[3].Nom := 'BT12';
	"DB_BIBLIOTHEQUE".Mobile[#index].Pos[3].Mob_Suiv[0] := "Index_Mobile"('BT12');

	"DB_BIBLIOTHEQUE".Mobile[#index].Tps_Asserv := t#1s;
	"DB_BIBLIOTHEQUE".Mobile[#index].Tps_Att := t#1s;
	"DB_BIBLIOTHEQUE".Mobile[#index].Tps_Arr := t#0s;
	"DB_BIBLIOTHEQUE".Mobile[#index].Tps_Vid := T#5s;
	"DB_BIBLIOTHEQUE".Mobile[#index].Tps_Chang_Pos := T#0s;

	// VERS BT10
	"DB_BIBLIOTHEQUE".Mobile[#index].Pos[0].Entr0_Ap_Pos[0] := "I_RP_REV01_BT17";
	"DB_BIBLIOTHEQUE".Mobile[#index].Pos[0].Entr0_Ap_Pos[1] := "I_RP_REV01_BT16";
	"DB_BIBLIOTHEQUE".Mobile[#index].Pos[0].Entr0_Ap_Pos[2] := "I_RP_REV01_BT12";
	"DB_BIBLIOTHEQUE".Mobile[#index].Pos[0].Entr1_Ap_Pos[0] := "I_RP_REV01_BT10";
	"DB_BIBLIOTHEQUE".Mobile[#index].Pos[0].Sort1[0] := "I_CM_REV01";
	"DB_BIBLIOTHEQUE".Mobile[#index].Pos[0].Sort1[1] := "I_FCP_REV01_BT10";
	"DB_BIBLIOTHEQUE".Mobile[#index].Pos[0].Sort0_Pr_Fin_Pos[0] := "I_CM_REV01";
	"DB_BIBLIOTHEQUE".Mobile[#index].Pos[0].Sort0_Pr_Fin_Pos[1] := "I_FCP_REV01_BT10";
	"DB_BIBLIOTHEQUE".Mobile[#index].Pos[0].Sort0_Ap_Pos[0] := "I_CM_REV01";
	// VERS BT17
	"DB_BIBLIOTHEQUE".Mobile[#index].Pos[1].Entr0_Ap_Pos[0] := "I_RP_REV01_BT10";
	"DB_BIBLIOTHEQUE".Mobile[#index].Pos[1].Entr0_Ap_Pos[1] := "I_RP_REV01_BT16";
	"DB_BIBLIOTHEQUE".Mobile[#index].Pos[1].Entr0_Ap_Pos[2] := "I_RP_REV01_BT12";
	"DB_BIBLIOTHEQUE".Mobile[#index].Pos[1].Entr1_Ap_Pos[0] := "I_RP_REV01_BT17";
	"DB_BIBLIOTHEQUE".Mobile[#index].Pos[1].Sort1[0] := "I_CM_REV01";
	"DB_BIBLIOTHEQUE".Mobile[#index].Pos[1].Sort1[1] := "I_FCP_REV01_BT17";
	"DB_BIBLIOTHEQUE".Mobile[#index].Pos[1].Sort0_Pr_Fin_Pos[0] := "I_CM_REV01";
	"DB_BIBLIOTHEQUE".Mobile[#index].Pos[1].Sort0_Pr_Fin_Pos[1] := "I_FCP_REV01_BT17";
	"DB_BIBLIOTHEQUE".Mobile[#index].Pos[1].Sort0_Ap_Pos[0] := "I_CM_REV01";
	//VERS BT16
	"DB_BIBLIOTHEQUE".Mobile[#index].Pos[2].Entr0_Ap_Pos[0] := "I_RP_REV01_BT10";
	"DB_BIBLIOTHEQUE".Mobile[#index].Pos[2].Entr0_Ap_Pos[1] := "I_RP_REV01_BT12";
	"DB_BIBLIOTHEQUE".Mobile[#index].Pos[2].Entr0_Ap_Pos[2] := "I_RP_REV01_BT17";
	"DB_BIBLIOTHEQUE".Mobile[#index].Pos[2].Entr1_Ap_Pos[0] := "I_RP_REV01_BT16";
	"DB_BIBLIOTHEQUE".Mobile[#index].Pos[2].Sort1[0] := "I_CM_REV01";
	"DB_BIBLIOTHEQUE".Mobile[#index].Pos[2].Sort1[1] := "I_FCP_REV01_BT16";
	"DB_BIBLIOTHEQUE".Mobile[#index].Pos[2].Sort0_Pr_Fin_Pos[0] := "I_CM_REV01";
	"DB_BIBLIOTHEQUE".Mobile[#index].Pos[2].Sort0_Pr_Fin_Pos[1] := "I_FCP_REV01_BT16";
	"DB_BIBLIOTHEQUE".Mobile[#index].Pos[2].Sort0_Ap_Pos[0] := "I_CM_REV01";
	//VERS BT12
	"DB_BIBLIOTHEQUE".Mobile[#index].Pos[3].Entr0_Ap_Pos[0] := "I_RP_REV01_BT10";
	"DB_BIBLIOTHEQUE".Mobile[#index].Pos[3].Entr0_Ap_Pos[1] := "I_RP_REV01_BT17";
	"DB_BIBLIOTHEQUE".Mobile[#index].Pos[3].Entr0_Ap_Pos[2] := "I_RP_REV01_BT16";
	"DB_BIBLIOTHEQUE".Mobile[#index].Pos[3].Entr1_Ap_Pos[0] := "I_RP_REV01_BT12";
	"DB_BIBLIOTHEQUE".Mobile[#index].Pos[3].Sort1[0] := "I_CM_REV01";
	"DB_BIBLIOTHEQUE".Mobile[#index].Pos[3].Sort1[1] := "I_FCP_REV01_BT12";
	"DB_BIBLIOTHEQUE".Mobile[#index].Pos[3].Sort0_Pr_Fin_Pos[0] := "I_CM_REV01";
	"DB_BIBLIOTHEQUE".Mobile[#index].Pos[3].Sort0_Pr_Fin_Pos[1] := "I_FCP_REV01_BT12";
	"DB_BIBLIOTHEQUE".Mobile[#index].Pos[3].Sort0_Ap_Pos[0] := "I_CM_REV01";
	#index := #index + 1;

	//++++++++++++++++++++++++++++++++++++++++++++++++++++++++++++++/*321*/
	"DB_BIBLIOTHEQUE".Mobile[#index].Nom := 'TRP_AV_BR1';
	"DB_BIBLIOTHEQUE".Mobile[#index].Pos[0].Nom := 'FERMETURE';
	"DB_BIBLIOTHEQUE".Mobile[#index].Pos[1].Nom := 'OUVERTURE';
	"DB_BIBLIOTHEQUE".Mobile[#index].Tjr_Desasservi := TRUE;
	"Init_Tps"(#index);

	//position fermeture
	"DB_BIBLIOTHEQUE".Mobile[#index].Pos[0].Entr0_Ap_Pos[0] := "I_RPO_TRP_TRM_BR1";
	"DB_BIBLIOTHEQUE".Mobile[#index].Pos[0].Entr1_Ap_Pos[0] := "I_RPF_TRP_TRM_BR1";
	"DB_BIBLIOTHEQUE".Mobile[#index].Pos[0].Sort0[0] := "I_CO_TRP_TRM_BR1";
	"DB_BIBLIOTHEQUE".Mobile[#index].Pos[0].Sort1_Pr_Fin_Pos[0] := "I_CO_TRP_TRM_BR1";

	//position ouverture
	"DB_BIBLIOTHEQUE".Mobile[#index].Pos[1].Entr0_Ap_Pos[0] := "I_RPF_TRP_TRM_BR1";
	"DB_BIBLIOTHEQUE".Mobile[#index].Pos[1].Entr1_Ap_Pos[0] := "I_RPO_TRP_TRM_BR1";
	"DB_BIBLIOTHEQUE".Mobile[#index].Pos[1].Sort1[0] := "I_CO_TRP_TRM_BR1";
	"DB_BIBLIOTHEQUE".Mobile[#index].Pos[1].Sort0_Pr_Fin_Pos[0] := "I_CO_TRP_TRM_BR1";

	#index := #index + 1;
	//++++++++++++++++++++++++++++++++++++++++++++++++++++++++++++++/*322*/
	"DB_BIBLIOTHEQUE".Mobile[#index].Nom := 'TRP_AV_BR2';
	"DB_BIBLIOTHEQUE".Mobile[#index].Pos[0].Nom := 'FERMETURE';
	"DB_BIBLIOTHEQUE".Mobile[#index].Pos[1].Nom := 'OUVERTURE';
	"DB_BIBLIOTHEQUE".Mobile[#index].Tjr_Desasservi := TRUE;
	"Init_Tps"(#index);

	//position fermeture
	"DB_BIBLIOTHEQUE".Mobile[#index].Pos[0].Entr0_Ap_Pos[0] := "I_RPO_TRP_TRM_BR2";
	"DB_BIBLIOTHEQUE".Mobile[#index].Pos[0].Entr1_Ap_Pos[0] := "I_RPF_TRP_TRM_BR2";
	"DB_BIBLIOTHEQUE".Mobile[#index].Pos[0].Sort0[0] := "I_CO_TRP_TRM_BR2";
	"DB_BIBLIOTHEQUE".Mobile[#index].Pos[0].Sort1_Pr_Fin_Pos[0] := "I_CO_TRP_TRM_BR2";

	//position ouverture
	"DB_BIBLIOTHEQUE".Mobile[#index].Pos[1].Entr0_Ap_Pos[0] := "I_RPF_TRP_TRM_BR2";
	"DB_BIBLIOTHEQUE".Mobile[#index].Pos[1].Entr1_Ap_Pos[0] := "I_RPO_TRP_TRM_BR2";
	"DB_BIBLIOTHEQUE".Mobile[#index].Pos[1].Sort1[0] := "I_CO_TRP_TRM_BR2";
	"DB_BIBLIOTHEQUE".Mobile[#index].Pos[1].Sort0_Pr_Fin_Pos[0] := "I_CO_TRP_TRM_BR2";
	#index := #index + 1;
	//++++++++++++++++++++++++++++++++++++++++++++++++++++++++++++++/*323*/
	"DB_BIBLIOTHEQUE".Mobile[#index].Nom := 'TRP1_TMEL';
	"DB_BIBLIOTHEQUE".Mobile[#index].Pos[0].Nom := 'FERMETURE';
	"DB_BIBLIOTHEQUE".Mobile[#index].Pos[1].Nom := 'OUVERTURE';
	"DB_BIBLIOTHEQUE".Mobile[#index].Tjr_Desasservi := TRUE;
	"Init_Tps"(#index);

	//position fermeture
	"DB_BIBLIOTHEQUE".Mobile[#index].Pos[0].Entr0_Ap_Pos[0] := "I_RPO_TRP1_TMEL1";
	"DB_BIBLIOTHEQUE".Mobile[#index].Pos[0].Entr1_Ap_Pos[0] := "I_RPF_TRP1_TMEL1";
	"DB_BIBLIOTHEQUE".Mobile[#index].Pos[0].Sort0[0] := "I_CO_TRP1_TMEL1";
	"DB_BIBLIOTHEQUE".Mobile[#index].Pos[0].Sort1_Pr_Fin_Pos[0] := "I_CO_TRP1_TMEL1";

	//position ouverture
	"DB_BIBLIOTHEQUE".Mobile[#index].Pos[1].Entr0_Ap_Pos[0] := "I_RPF_TRP1_TMEL1";
	"DB_BIBLIOTHEQUE".Mobile[#index].Pos[1].Entr1_Ap_Pos[0] := "I_RPO_TRP1_TMEL1";
	"DB_BIBLIOTHEQUE".Mobile[#index].Pos[1].Sort1[0] := "I_CO_TRP1_TMEL1";
	"DB_BIBLIOTHEQUE".Mobile[#index].Pos[1].Sort0_Pr_Fin_Pos[0] := "I_CO_TRP1_TMEL1";
	#index := #index + 1;
	//++++++++++++++++++++++++++++++++++++++++++++++++++++++++++++++/*324*/
	"DB_BIBLIOTHEQUE".Mobile[#index].Nom := 'TMEL';
	"DB_BIBLIOTHEQUE".Mobile[#index].Pos[0].Nom := 'VID';
	"DB_BIBLIOTHEQUE".Mobile[#index].Tjr_Desasservi := TRUE;
	"Init_Tps"(#index);
	#index := #index + 1;
	//++++++++++++++++++++++++++++++++++++++++++++++++++++++++++++++/*325*/
	"DB_BIBLIOTHEQUE".Mobile[#index].Nom := 'MLG1';
	// "DB_BIBLIOTHEQUE".Mobile[#index].Mob_Suiv[0] := "Index_Mobile"('TMEL');
	// "DB_BIBLIOTHEQUE".Mobile[#index].Pos[0].Nom := 'DROITE';
	// "DB_BIBLIOTHEQUE".Mobile[#index].Pos[0].Mob_Suiv[0] := "Index_Mobile"('TMEL');
	"DB_BIBLIOTHEQUE".Mobile[#index].Tjr_Desasservi := TRUE;
	"DB_BIBLIOTHEQUE".Mobile[#index].Tps_Att := t#500ms;
	"DB_BIBLIOTHEQUE".Mobile[#index].Tps_Arr := t#0ms;

	"DB_BIBLIOTHEQUE".Mobile[#index].Tps_Max_Mar_Forc := t#0ms;
	"DB_BIBLIOTHEQUE".Mobile[#index].Tps_Vid := t#0ms;

	// Entrées avant pos
	"DB_BIBLIOTHEQUE".Mobile[#index].Pos[0].Entr0_Av_Pos[0] := "I_RD_DISJ_MEL1";
	// Entrées apres pos
	"DB_BIBLIOTHEQUE".Mobile[#index].Pos[0].Entr0_Ap_Pos[0] := "I_RD_DISJ_MEL1";
	"DB_BIBLIOTHEQUE".Mobile[#index].Pos[0].Entr1_Ap_Pos[0] := "I_RM_MEL1";

	// Entrées fin pos
	"DB_BIBLIOTHEQUE".Mobile[#index].Pos[0].Entr0_Ap_Fin_Pos[0] := "I_RM_MEL1";

	// Sorties
	"DB_BIBLIOTHEQUE".Mobile[#index].Pos[0].Sort1[0] := "I_CM_MEL1";
	"DB_BIBLIOTHEQUE".Mobile[#index].Pos[0].Sort0_Pr_Fin_Pos[0] := "I_CM_MEL1";
	#index := #index + 1;
	//++++++++++++++++++++++++++++++++++++++++++++++++++++++++++++++/*326*/
	"DB_BIBLIOTHEQUE".Mobile[#index].Nom := 'TRP1_MLG1';
	"DB_BIBLIOTHEQUE".Mobile[#index].Pos[0].Nom := 'OUVERTURE';
	"DB_BIBLIOTHEQUE".Mobile[#index].Pos[1].Nom := 'FERMETURE';
	"DB_BIBLIOTHEQUE".Mobile[#index].Tjr_Desasservi := TRUE;
	"Init_Tps"(#index);

	//position fermeture
	"DB_BIBLIOTHEQUE".Mobile[#index].Pos[0].Entr0_Ap_Pos[0] := "I_RPO_TRP1_MLG";
	"DB_BIBLIOTHEQUE".Mobile[#index].Pos[0].Entr1_Ap_Pos[0] := "I_RPF_TRP1_MLG";
	"DB_BIBLIOTHEQUE".Mobile[#index].Pos[0].Sort0[0] := "I_CO_TRP1_MLG1";
	"DB_BIBLIOTHEQUE".Mobile[#index].Pos[0].Sort1_Pr_Fin_Pos[0] := "I_CO_TRP1_MLG1";
	//position fermeture
	"DB_BIBLIOTHEQUE".Mobile[#index].Pos[0].Entr0_Ap_Pos[1] := "I_RPO_TRP1_MLG";
	"DB_BIBLIOTHEQUE".Mobile[#index].Pos[0].Entr1_Ap_Pos[1] := "I_RPF_TRP1_MLG";
	"DB_BIBLIOTHEQUE".Mobile[#index].Pos[0].Sort0[1] := "I_CO_TRP1_MLG1";
	"DB_BIBLIOTHEQUE".Mobile[#index].Pos[0].Sort1_Pr_Fin_Pos[1] := "I_CO_TRP1_MLG1";
	//position ouverture
	"DB_BIBLIOTHEQUE".Mobile[#index].Pos[1].Entr0_Ap_Pos[0] := "I_RPF_TRP1_MLG";
	"DB_BIBLIOTHEQUE".Mobile[#index].Pos[1].Entr1_Ap_Pos[0] := "I_RPO_TRP1_MLG";
	"DB_BIBLIOTHEQUE".Mobile[#index].Pos[1].Sort1[0] := "I_CO_TRP1_MLG1";
	"DB_BIBLIOTHEQUE".Mobile[#index].Pos[1].Sort0_Pr_Fin_Pos[0] := "I_CO_TRP1_MLG1";
	//position ouverture
	"DB_BIBLIOTHEQUE".Mobile[#index].Pos[1].Entr0_Ap_Pos[1] := "I_RPF_TRP1_MLG";
	"DB_BIBLIOTHEQUE".Mobile[#index].Pos[1].Entr1_Ap_Pos[0] := "I_RPO_TRP1_MLG";
	"DB_BIBLIOTHEQUE".Mobile[#index].Pos[1].Sort1[1] := "I_CO_TRP1_MLG1";
	"DB_BIBLIOTHEQUE".Mobile[#index].Pos[1].Sort0_Pr_Fin_Pos[1] := "I_CO_TRP1_MLG1";
	#index := #index + 1;
	//++++++++++++++++++++++++++++++++++++++++++++++++++++++++++++++/*327*/
	"DB_BIBLIOTHEQUE".Mobile[#index].Nom := 'TRP2_T29';
	"DB_BIBLIOTHEQUE".Mobile[#index].Mob_Suiv[0] := "Index_Mobile"('SBP3');
	"DB_BIBLIOTHEQUE".Mobile[#index].Pos[0].Nom := 'FERMETURE';
	"DB_BIBLIOTHEQUE".Mobile[#index].Pos[0].Mob_Suiv[0] := "Index_Mobile"('SBP3');
	"DB_BIBLIOTHEQUE".Mobile[#index].Pos[1].Nom := 'OUVERTURE';
	"DB_BIBLIOTHEQUE".Mobile[#index].Pos[1].Mob_Suiv[0] := "Index_Mobile"('SBP3');

	//position fermeture
	"DB_BIBLIOTHEQUE".Mobile[#index].Pos[0].Entr0_Ap_Pos[0] := "I_RPO_TRP2T29";
	"DB_BIBLIOTHEQUE".Mobile[#index].Pos[0].Entr1_Ap_Pos[0] := "I_RPF_TRP2T29";
	"DB_BIBLIOTHEQUE".Mobile[#index].Pos[0].Sort0[0] := "I_CO_TRP2T29";
	"DB_BIBLIOTHEQUE".Mobile[#index].Pos[0].Sort0_Pr_Fin_Pos[0] := "I_CO_TRP2T29";

	//position ouverture
	"DB_BIBLIOTHEQUE".Mobile[#index].Pos[1].Entr0_Ap_Pos[0] := "I_RPF_TRP2T29";
	"DB_BIBLIOTHEQUE".Mobile[#index].Pos[1].Entr1_Ap_Pos[0] := "I_RPO_TRP2T29";
	"DB_BIBLIOTHEQUE".Mobile[#index].Pos[1].Sort1[0] := "I_CO_TRP2T29";
	"DB_BIBLIOTHEQUE".Mobile[#index].Pos[1].Sort0_Pr_Fin_Pos[0] := "I_CO_TRP2T29";
	"Init_Tps"(#index);
	#index := #index + 1;
	//++++++++++++++++++++++++++++++++++++++++++++++++++++++++++++++/*328*/
	"DB_BIBLIOTHEQUE".Mobile[#index].Nom := 'PMP_LIQ1';
	"DB_BIBLIOTHEQUE".Mobile[#index].Mob_Suiv[0] := "Index_Mobile"('VN1_MLG1');
	"DB_BIBLIOTHEQUE".Mobile[#index].Mob_Suiv[1] := "Index_Mobile"('VN1_MLG2');
	"DB_BIBLIOTHEQUE".Mobile[#index].Pos[0].Nom := 'VERS_MLG1';
	"DB_BIBLIOTHEQUE".Mobile[#index].Pos[0].Suiv_Enc := "Index_Mobile"('VN1_MLG1');
	"DB_BIBLIOTHEQUE".Mobile[#index].Pos[1].Nom := 'VERS_MLG2';
	"DB_BIBLIOTHEQUE".Mobile[#index].Pos[1].Suiv_Enc := "Index_Mobile"('VN1_MLG2');
	"Init_Tps"(#index);

	// Entrées avant pos
	"DB_BIBLIOTHEQUE".Mobile[#index].Pos[0].Entr0_Av_Pos[0] := "I_RD_DISJ_PMP1";
	// Entrées apres pos
	"DB_BIBLIOTHEQUE".Mobile[#index].Pos[0].Entr0_Ap_Pos[0] := "I_RD_DISJ_PMP1";
	"DB_BIBLIOTHEQUE".Mobile[#index].Pos[0].Entr1_Ap_Pos[0] := "I_RM_PMP1";
	// Entrées fin pos
	"DB_BIBLIOTHEQUE".Mobile[#index].Pos[0].Entr0_Ap_Fin_Pos[0] := "I_RM_PMP1";
	// Sorties
	"DB_BIBLIOTHEQUE".Mobile[#index].Pos[0].Sort1[0] := "I_CM_POMPE01";
	"DB_BIBLIOTHEQUE".Mobile[#index].Pos[0].Sort0_Pr_Fin_Pos[0] := "I_CM_POMPE01";

	// Entrées avant pos
	"DB_BIBLIOTHEQUE".Mobile[#index].Pos[1].Entr0_Av_Pos[0] := "I_RD_DISJ_PMP1";
	// Entrées apres pos
	"DB_BIBLIOTHEQUE".Mobile[#index].Pos[1].Entr0_Ap_Pos[0] := "I_RD_DISJ_PMP1";
	"DB_BIBLIOTHEQUE".Mobile[#index].Pos[1].Entr1_Ap_Pos[0] := "I_RM_PMP1";
	// Entrées fin pos
	"DB_BIBLIOTHEQUE".Mobile[#index].Pos[1].Entr0_Ap_Fin_Pos[0] := "I_RM_PMP1";
	// Sorties
	"DB_BIBLIOTHEQUE".Mobile[#index].Pos[1].Sort1[0] := "I_CM_POMPE01";
	"DB_BIBLIOTHEQUE".Mobile[#index].Pos[1].Sort0_Pr_Fin_Pos[0] := "I_CM_POMPE01";
	#index := #index + 1;
	//++++++++++++++++++++++++++++++++++++++++++++++++++++++++++++++/*329*/
	"DB_BIBLIOTHEQUE".Mobile[#index].Nom := 'PMP_LIQ2';
	"DB_BIBLIOTHEQUE".Mobile[#index].Mob_Suiv[0] := "Index_Mobile"('VN2_MLG1');
	"DB_BIBLIOTHEQUE".Mobile[#index].Mob_Suiv[1] := "Index_Mobile"('VN2_MLG2');
	"DB_BIBLIOTHEQUE".Mobile[#index].Pos[0].Nom := 'VERS_MLG1';
	"DB_BIBLIOTHEQUE".Mobile[#index].Pos[0].Suiv_Enc := "Index_Mobile"('VN2_MLG1');
	"DB_BIBLIOTHEQUE".Mobile[#index].Pos[1].Nom := 'VERS_MLG2';
	"DB_BIBLIOTHEQUE".Mobile[#index].Pos[1].Suiv_Enc := "Index_Mobile"('VN2_MLG2');
	"Init_Tps"(#index);

	// Entrées avant pos
	"DB_BIBLIOTHEQUE".Mobile[#index].Pos[0].Entr0_Av_Pos[0] := "I_RD_DISJ_PMP2";
	// Entrées apres pos
	"DB_BIBLIOTHEQUE".Mobile[#index].Pos[0].Entr0_Ap_Pos[0] := "I_RD_DISJ_PMP2";
	"DB_BIBLIOTHEQUE".Mobile[#index].Pos[0].Entr1_Ap_Pos[0] := "I_RM_PMP2";
	// Entrées fin pos
	"DB_BIBLIOTHEQUE".Mobile[#index].Pos[0].Entr0_Ap_Fin_Pos[0] := "I_RM_PMP2";
	// Sorties
	"DB_BIBLIOTHEQUE".Mobile[#index].Pos[0].Sort1[0] := "I_CM_POMPE02";
	"DB_BIBLIOTHEQUE".Mobile[#index].Pos[0].Sort0_Pr_Fin_Pos[0] := "I_CM_POMPE02";


	// Entrées avant pos
	"DB_BIBLIOTHEQUE".Mobile[#index].Pos[1].Entr0_Av_Pos[0] := "I_RD_DISJ_PMP2";
	// Entrées apres pos
	"DB_BIBLIOTHEQUE".Mobile[#index].Pos[1].Entr0_Ap_Pos[0] := "I_RD_DISJ_PMP2";
	"DB_BIBLIOTHEQUE".Mobile[#index].Pos[1].Entr1_Ap_Pos[0] := "I_RM_PMP2";
	// Entrées fin pos
	"DB_BIBLIOTHEQUE".Mobile[#index].Pos[1].Entr0_Ap_Fin_Pos[0] := "I_RM_PMP2";
	// Sorties
	"DB_BIBLIOTHEQUE".Mobile[#index].Pos[1].Sort1[0] := "I_CM_POMPE02";
	"DB_BIBLIOTHEQUE".Mobile[#index].Pos[1].Sort0_Pr_Fin_Pos[0] := "I_CM_POMPE02";
	#index := #index + 1;
	//++++++++++++++++++++++++++++++++++++++++++++++++++++++++++++++/*330*/
	"DB_BIBLIOTHEQUE".Mobile[#index].Nom := 'PMP_LIQ3';
	"DB_BIBLIOTHEQUE".Mobile[#index].Mob_Suiv[0] := "Index_Mobile"('VN3_MLG1');
	"DB_BIBLIOTHEQUE".Mobile[#index].Mob_Suiv[1] := "Index_Mobile"('VN3_MLG2');
	"DB_BIBLIOTHEQUE".Mobile[#index].Pos[0].Nom := 'VERS_MLG1';
	"DB_BIBLIOTHEQUE".Mobile[#index].Pos[0].Suiv_Enc := "Index_Mobile"('VN3_MLG1');
	"DB_BIBLIOTHEQUE".Mobile[#index].Pos[1].Nom := 'VERS_MLG2';
	"DB_BIBLIOTHEQUE".Mobile[#index].Pos[1].Suiv_Enc := "Index_Mobile"('VN3_MLG2');
	"Init_Tps"(#index);

	// Entrées avant pos
	"DB_BIBLIOTHEQUE".Mobile[#index].Pos[0].Entr0_Av_Pos[0] := "I_RD_DISJ_PMP3";
	// Entrées apres pos
	"DB_BIBLIOTHEQUE".Mobile[#index].Pos[0].Entr0_Ap_Pos[0] := "I_RD_DISJ_PMP3";
	"DB_BIBLIOTHEQUE".Mobile[#index].Pos[0].Entr1_Ap_Pos[0] := "I_RM_PMP3";
	// Entrées fin pos
	"DB_BIBLIOTHEQUE".Mobile[#index].Pos[0].Entr0_Ap_Fin_Pos[0] := "I_RM_PMP3";
	// Sorties
	"DB_BIBLIOTHEQUE".Mobile[#index].Pos[0].Sort1[0] := "I_CM_POMPE03";
	"DB_BIBLIOTHEQUE".Mobile[#index].Pos[0].Sort0_Pr_Fin_Pos[0] := "I_CM_POMPE03";



	// Entrées avant pos
	"DB_BIBLIOTHEQUE".Mobile[#index].Pos[1].Entr0_Av_Pos[0] := "I_RD_DISJ_PMP3";
	// Entrées apres pos
	"DB_BIBLIOTHEQUE".Mobile[#index].Pos[1].Entr0_Ap_Pos[0] := "I_RD_DISJ_PMP3";
	"DB_BIBLIOTHEQUE".Mobile[#index].Pos[1].Entr1_Ap_Pos[0] := "I_RM_PMP3";
	// Entrées fin pos
	"DB_BIBLIOTHEQUE".Mobile[#index].Pos[1].Entr0_Ap_Fin_Pos[0] := "I_RM_PMP3";
	// Sorties
	"DB_BIBLIOTHEQUE".Mobile[#index].Pos[1].Sort1[0] := "I_CM_POMPE03";
	"DB_BIBLIOTHEQUE".Mobile[#index].Pos[1].Sort0_Pr_Fin_Pos[0] := "I_CM_POMPE03";
	#index := #index + 1;
	//++++++++++++++++++++++++++++++++++++++++++++++++++++++++++++++/*331*/
	"DB_BIBLIOTHEQUE".Mobile[#index].Nom := 'PMP_LIQ4';
	"DB_BIBLIOTHEQUE".Mobile[#index].Mob_Suiv[0] := "Index_Mobile"('VN4_MLG1');
	"DB_BIBLIOTHEQUE".Mobile[#index].Mob_Suiv[1] := "Index_Mobile"('VN4_MLG2');
	"DB_BIBLIOTHEQUE".Mobile[#index].Pos[0].Nom := 'VERS_MLG1';
	"DB_BIBLIOTHEQUE".Mobile[#index].Pos[0].Suiv_Enc := "Index_Mobile"('VN4_MLG1');
	"DB_BIBLIOTHEQUE".Mobile[#index].Pos[1].Nom := 'VERS_MLG2';
	"DB_BIBLIOTHEQUE".Mobile[#index].Pos[1].Suiv_Enc := "Index_Mobile"('VN4_MLG2');
	"Init_Tps"(#index);

	// Entrées avant pos
	"DB_BIBLIOTHEQUE".Mobile[#index].Pos[0].Entr0_Av_Pos[0] := "I_RD_DISJ_PMP4";
	// Entrées apres pos
	"DB_BIBLIOTHEQUE".Mobile[#index].Pos[0].Entr0_Ap_Pos[0] := "I_RD_DISJ_PMP4";
	"DB_BIBLIOTHEQUE".Mobile[#index].Pos[0].Entr1_Ap_Pos[0] := "I_RM_PMP4";
	// Entrées fin pos
	"DB_BIBLIOTHEQUE".Mobile[#index].Pos[0].Entr0_Ap_Fin_Pos[0] := "I_RM_PMP4";
	// Sorties
	"DB_BIBLIOTHEQUE".Mobile[#index].Pos[0].Sort1[0] := "I_CM_POMPE04";
	"DB_BIBLIOTHEQUE".Mobile[#index].Pos[0].Sort0_Pr_Fin_Pos[0] := "I_CM_POMPE04";


	// Entrées avant pos
	"DB_BIBLIOTHEQUE".Mobile[#index].Pos[1].Entr0_Av_Pos[0] := "I_RD_DISJ_PMP4";
	// Entrées apres pos
	"DB_BIBLIOTHEQUE".Mobile[#index].Pos[1].Entr0_Ap_Pos[0] := "I_RD_DISJ_PMP4";
	"DB_BIBLIOTHEQUE".Mobile[#index].Pos[1].Entr1_Ap_Pos[0] := "I_RM_PMP4";
	// Entrées fin pos
	"DB_BIBLIOTHEQUE".Mobile[#index].Pos[1].Entr0_Ap_Fin_Pos[0] := "I_RM_PMP4";
	// Sorties
	"DB_BIBLIOTHEQUE".Mobile[#index].Pos[1].Sort1[0] := "I_CM_POMPE04";
	"DB_BIBLIOTHEQUE".Mobile[#index].Pos[1].Sort0_Pr_Fin_Pos[0] := "I_CM_POMPE04";
	#index := #index + 1;
	//++++++++++++++++++++++++++++++++++++++++++++++++++++++++++++++/*332*/
	"DB_BIBLIOTHEQUE".Mobile[#index].Nom := 'PMP_LIQ5';
	"DB_BIBLIOTHEQUE".Mobile[#index].Mob_Suiv[0] := "Index_Mobile"('VN5_MLG1');
	"DB_BIBLIOTHEQUE".Mobile[#index].Mob_Suiv[1] := "Index_Mobile"('VN5_MLG2');
	"DB_BIBLIOTHEQUE".Mobile[#index].Pos[0].Nom := 'VERS_MLG1';
	"DB_BIBLIOTHEQUE".Mobile[#index].Pos[0].Suiv_Enc := "Index_Mobile"('VN5_MLG1');
	"DB_BIBLIOTHEQUE".Mobile[#index].Pos[1].Nom := 'VERS_MLG2';
	"DB_BIBLIOTHEQUE".Mobile[#index].Pos[1].Suiv_Enc := "Index_Mobile"('VN5_MLG2');
	"Init_Tps"(#index);

	// Entrées avant pos
	"DB_BIBLIOTHEQUE".Mobile[#index].Pos[0].Entr0_Av_Pos[0] := "I_RD_DISJ_PMP5";
	// Entrées apres pos
	"DB_BIBLIOTHEQUE".Mobile[#index].Pos[0].Entr0_Ap_Pos[0] := "I_RD_DISJ_PMP5";
	"DB_BIBLIOTHEQUE".Mobile[#index].Pos[0].Entr1_Ap_Pos[0] := "I_RM_PMP5";
	// Entrées fin pos
	"DB_BIBLIOTHEQUE".Mobile[#index].Pos[0].Entr0_Ap_Fin_Pos[0] := "I_RM_PMP5";
	// Sorties
	"DB_BIBLIOTHEQUE".Mobile[#index].Pos[0].Sort1[0] := "I_CM_POMPE05";
	"DB_BIBLIOTHEQUE".Mobile[#index].Pos[0].Sort0_Pr_Fin_Pos[0] := "I_CM_POMPE05";



	// Entrées avant pos
	"DB_BIBLIOTHEQUE".Mobile[#index].Pos[1].Entr0_Av_Pos[0] := "I_RD_DISJ_PMP5";
	// Entrées apres pos
	"DB_BIBLIOTHEQUE".Mobile[#index].Pos[1].Entr0_Ap_Pos[0] := "I_RD_DISJ_PMP5";
	"DB_BIBLIOTHEQUE".Mobile[#index].Pos[1].Entr1_Ap_Pos[0] := "I_RM_PMP5";
	// Entrées fin pos
	"DB_BIBLIOTHEQUE".Mobile[#index].Pos[1].Entr0_Ap_Fin_Pos[0] := "I_RM_PMP5";
	// Sorties
	"DB_BIBLIOTHEQUE".Mobile[#index].Pos[1].Sort1[0] := "I_CM_POMPE05";
	"DB_BIBLIOTHEQUE".Mobile[#index].Pos[1].Sort0_Pr_Fin_Pos[0] := "I_CM_POMPE05";
	#index := #index + 1;
	//++++++++++++++++++++++++++++++++++++++++++++++++++++++++++++++/*333*/
	"DB_BIBLIOTHEQUE".Mobile[#index].Nom := 'VN1_MLG1';
	"DB_BIBLIOTHEQUE".Mobile[#index].Pos[0].Nom := 'FERMETURE';
	"DB_BIBLIOTHEQUE".Mobile[#index].Pos[1].Nom := 'OUVERTURE';
	"DB_BIBLIOTHEQUE".Mobile[#index].Tjr_Desasservi := TRUE;
	"DB_BIBLIOTHEQUE".Mobile[#index].Tps_Att := t#500ms;
	"DB_BIBLIOTHEQUE".Mobile[#index].Tps_Arr := t#0ms;

	//position fermeture
	"DB_BIBLIOTHEQUE".Mobile[#index].Pos[0].Entr0_Ap_Pos[0] := "I_RPO_VPMP1_MLG1";
	"DB_BIBLIOTHEQUE".Mobile[#index].Pos[0].Entr1_Ap_Pos[0] := "I_RPF_VPMP1_MLG1";
	"DB_BIBLIOTHEQUE".Mobile[#index].Pos[0].Sort0[0] := "I_CO_VPMP1_MLG1";
	"DB_BIBLIOTHEQUE".Mobile[#index].Pos[0].Sort0_Pr_Fin_Pos[0] := "I_CO_VPMP1_MLG1";

	//position ouverture
	//Verouillage
	"DB_BIBLIOTHEQUE".Mobile[#index].Pos[1].Entr1_Av_Pos[0] := "I_RPF_VPMP1_MLG1";
	"DB_BIBLIOTHEQUE".Mobile[#index].Pos[1].Entr0_Ap_Pos[0] := "I_RPF_VPMP1_MLG1";
	"DB_BIBLIOTHEQUE".Mobile[#index].Pos[1].Entr1_Ap_Pos[0] := "I_RPO_VPMP1_MLG1";
	"DB_BIBLIOTHEQUE".Mobile[#index].Pos[1].Sort1[0] := "I_CO_VPMP1_MLG1";
	"DB_BIBLIOTHEQUE".Mobile[#index].Pos[1].Sort0_Pr_Fin_Pos[0] := "I_CO_VPMP1_MLG1";
	#index := #index + 1;
	//++++++++++++++++++++++++++++++++++++++++++++++++++++++++++++++/*334*/
	"DB_BIBLIOTHEQUE".Mobile[#index].Nom := 'VN2_MLG1';
	"DB_BIBLIOTHEQUE".Mobile[#index].Pos[0].Nom := 'FERMETURE';
	"DB_BIBLIOTHEQUE".Mobile[#index].Pos[1].Nom := 'OUVERTURE';
	"DB_BIBLIOTHEQUE".Mobile[#index].Tjr_Desasservi := TRUE;
	"Init_Tps"(#index);

	//position fermeture
	"DB_BIBLIOTHEQUE".Mobile[#index].Pos[0].Entr0_Ap_Pos[0] := "I_RPO_VPMP2_MLG1";
	"DB_BIBLIOTHEQUE".Mobile[#index].Pos[0].Entr1_Ap_Pos[0] := "I_RPF_VPMP2_MLG1";
	"DB_BIBLIOTHEQUE".Mobile[#index].Pos[0].Sort0[0] := "I_CO_VPMP2_MLG1";
	"DB_BIBLIOTHEQUE".Mobile[#index].Pos[0].Sort0_Pr_Fin_Pos[0] := "I_CO_VPMP2_MLG1";

	//position ouverture
	//Verouillage
	"DB_BIBLIOTHEQUE".Mobile[#index].Pos[1].Entr1_Av_Pos[0] := "I_RPF_VPMP2_MLG1";
	"DB_BIBLIOTHEQUE".Mobile[#index].Pos[1].Entr0_Ap_Pos[0] := "I_RPF_VPMP2_MLG1";
	"DB_BIBLIOTHEQUE".Mobile[#index].Pos[1].Entr1_Ap_Pos[0] := "I_RPO_VPMP2_MLG1";
	"DB_BIBLIOTHEQUE".Mobile[#index].Pos[1].Sort1[0] := "I_CO_VPMP2_MLG1";
	"DB_BIBLIOTHEQUE".Mobile[#index].Pos[1].Sort0_Pr_Fin_Pos[0] := "I_CO_VPMP2_MLG1";
	#index := #index + 1;
	//++++++++++++++++++++++++++++++++++++++++++++++++++++++++++++++/*335*/
	"DB_BIBLIOTHEQUE".Mobile[#index].Nom := 'VN3_MLG1';
	"DB_BIBLIOTHEQUE".Mobile[#index].Pos[0].Nom := 'FERMETURE';
	"DB_BIBLIOTHEQUE".Mobile[#index].Pos[1].Nom := 'OUVERTURE';
	"DB_BIBLIOTHEQUE".Mobile[#index].Tjr_Desasservi := TRUE;
	"Init_Tps"(#index);

	//position fermeture
	"DB_BIBLIOTHEQUE".Mobile[#index].Pos[0].Entr0_Ap_Pos[0] := "I_RPO_VPMP3_MLG1";
	"DB_BIBLIOTHEQUE".Mobile[#index].Pos[0].Entr1_Ap_Pos[0] := "I_RPF_VPMP3_MLG1";
	"DB_BIBLIOTHEQUE".Mobile[#index].Pos[0].Sort0[0] := "I_CO_VPMP3_MLG1";
	"DB_BIBLIOTHEQUE".Mobile[#index].Pos[0].Sort0_Pr_Fin_Pos[0] := "I_CO_VPMP3_MLG1";

	//position ouverture
	//Verouillage
	"DB_BIBLIOTHEQUE".Mobile[#index].Pos[1].Entr1_Av_Pos[0] := "I_RPF_VPMP3_MLG1";
	"DB_BIBLIOTHEQUE".Mobile[#index].Pos[1].Entr0_Ap_Pos[0] := "I_RPF_VPMP3_MLG1";
	"DB_BIBLIOTHEQUE".Mobile[#index].Pos[1].Entr1_Ap_Pos[0] := "I_RPO_VPMP3_MLG1";
	"DB_BIBLIOTHEQUE".Mobile[#index].Pos[1].Sort1[0] := "I_CO_VPMP3_MLG1";
	"DB_BIBLIOTHEQUE".Mobile[#index].Pos[1].Sort0_Pr_Fin_Pos[0] := "I_CO_VPMP3_MLG1";
	#index := #index + 1;
	//++++++++++++++++++++++++++++++++++++++++++++++++++++++++++++++/*336*/
	"DB_BIBLIOTHEQUE".Mobile[#index].Nom := 'VN4_MLG1';
	"DB_BIBLIOTHEQUE".Mobile[#index].Pos[0].Nom := 'FERMETURE';
	"DB_BIBLIOTHEQUE".Mobile[#index].Pos[1].Nom := 'OUVERTURE';
	"DB_BIBLIOTHEQUE".Mobile[#index].Tjr_Desasservi := TRUE;
	"Init_Tps"(#index);

	//position fermeture
	"DB_BIBLIOTHEQUE".Mobile[#index].Pos[0].Entr0_Ap_Pos[0] := "I_RPO_VPMP4_MLG1";
	"DB_BIBLIOTHEQUE".Mobile[#index].Pos[0].Entr1_Ap_Pos[0] := "I_RPF_VPMP4_MLG1";
	"DB_BIBLIOTHEQUE".Mobile[#index].Pos[0].Sort0[0] := "I_CO_VPMP4_MLG1";
	"DB_BIBLIOTHEQUE".Mobile[#index].Pos[0].Sort0_Pr_Fin_Pos[0] := "I_CO_VPMP4_MLG1";

	//position ouverture
	//Verouillage
	"DB_BIBLIOTHEQUE".Mobile[#index].Pos[1].Entr1_Av_Pos[0] := "I_RPF_VPMP4_MLG1";
	"DB_BIBLIOTHEQUE".Mobile[#index].Pos[1].Entr0_Ap_Pos[0] := "I_RPF_VPMP4_MLG1";
	"DB_BIBLIOTHEQUE".Mobile[#index].Pos[1].Entr1_Ap_Pos[0] := "I_RPO_VPMP4_MLG1";
	"DB_BIBLIOTHEQUE".Mobile[#index].Pos[1].Sort1[0] := "I_CO_VPMP4_MLG1";
	"DB_BIBLIOTHEQUE".Mobile[#index].Pos[1].Sort0_Pr_Fin_Pos[0] := "I_CO_VPMP4_MLG1";
	#index := #index + 1;
	//++++++++++++++++++++++++++++++++++++++++++++++++++++++++++++++/*337*/
	"DB_BIBLIOTHEQUE".Mobile[#index].Nom := 'VN5_MLG1';
	"DB_BIBLIOTHEQUE".Mobile[#index].Pos[0].Nom := 'FERMETURE';
	"DB_BIBLIOTHEQUE".Mobile[#index].Pos[1].Nom := 'OUVERTURE';
	"DB_BIBLIOTHEQUE".Mobile[#index].Tjr_Desasservi := TRUE;
	"Init_Tps"(#index);

	//position fermeture
	"DB_BIBLIOTHEQUE".Mobile[#index].Pos[0].Entr0_Ap_Pos[0] := "I_RPO_VPMP5_MLG1";
	"DB_BIBLIOTHEQUE".Mobile[#index].Pos[0].Entr1_Ap_Pos[0] := "I_RPF_VPMP5_MLG1";
	"DB_BIBLIOTHEQUE".Mobile[#index].Pos[0].Sort0[0] := "I_CO_VPMP5_MLG1";
	"DB_BIBLIOTHEQUE".Mobile[#index].Pos[0].Sort0_Pr_Fin_Pos[0] := "I_CO_VPMP5_MLG1";

	//position ouverture
	//Verouillage
	"DB_BIBLIOTHEQUE".Mobile[#index].Pos[1].Entr1_Av_Pos[0] := "I_RPF_VPMP5_MLG1";
	"DB_BIBLIOTHEQUE".Mobile[#index].Pos[1].Entr0_Ap_Pos[0] := "I_RPF_VPMP5_MLG1";
	"DB_BIBLIOTHEQUE".Mobile[#index].Pos[1].Entr1_Ap_Pos[0] := "I_RPO_VPMP5_MLG1";
	"DB_BIBLIOTHEQUE".Mobile[#index].Pos[1].Sort1[0] := "I_CO_VPMP5_MLG1";
	"DB_BIBLIOTHEQUE".Mobile[#index].Pos[1].Sort0_Pr_Fin_Pos[0] := "I_CO_VPMP5_MLG1";
	#index := #index + 1;
	//++++++++++++++++++++++++++++++++++++++++++++++++++++++++++++++/*338*/
	"DB_BIBLIOTHEQUE".Mobile[#index].Nom := 'VN1_MLG2';
	"DB_BIBLIOTHEQUE".Mobile[#index].Pos[0].Nom := 'FERMETURE';
	"DB_BIBLIOTHEQUE".Mobile[#index].Pos[1].Nom := 'OUVERTURE';
	"DB_BIBLIOTHEQUE".Mobile[#index].Tjr_Desasservi := TRUE;
	"Init_Tps"(#index);

	//position fermeture
	"DB_BIBLIOTHEQUE".Mobile[#index].Pos[0].Entr0_Ap_Pos[0] := "I_RPO_VPMP1_MLG2";
	"DB_BIBLIOTHEQUE".Mobile[#index].Pos[0].Entr1_Ap_Pos[0] := "I_RPF_VPMP1_MLG2";
	"DB_BIBLIOTHEQUE".Mobile[#index].Pos[0].Sort0[0] := "I_CO_VPMP1_MLG2";
	"DB_BIBLIOTHEQUE".Mobile[#index].Pos[0].Sort0_Pr_Fin_Pos[0] := "I_CO_VPMP1_MLG2";

	//position ouverture
	//Verouillage
	"DB_BIBLIOTHEQUE".Mobile[#index].Pos[1].Entr1_Av_Pos[0] := "I_RPF_VPMP1_MLG2";
	"DB_BIBLIOTHEQUE".Mobile[#index].Pos[1].Entr0_Ap_Pos[0] := "I_RPF_VPMP1_MLG2";
	"DB_BIBLIOTHEQUE".Mobile[#index].Pos[1].Entr1_Ap_Pos[0] := "I_RPO_VPMP1_MLG2";
	"DB_BIBLIOTHEQUE".Mobile[#index].Pos[1].Sort1[0] := "I_CO_VPMP1_MLG2";
	"DB_BIBLIOTHEQUE".Mobile[#index].Pos[1].Sort0_Pr_Fin_Pos[0] := "I_CO_VPMP1_MLG2";
	#index := #index + 1;
	//++++++++++++++++++++++++++++++++++++++++++++++++++++++++++++++/*339*/
	"DB_BIBLIOTHEQUE".Mobile[#index].Nom := 'VN2_MLG2';
	"DB_BIBLIOTHEQUE".Mobile[#index].Pos[0].Nom := 'FERMETURE';
	"DB_BIBLIOTHEQUE".Mobile[#index].Pos[1].Nom := 'OUVERTURE';
	"DB_BIBLIOTHEQUE".Mobile[#index].Tjr_Desasservi := TRUE;
	"Init_Tps"(#index);

	//position fermeture
	"DB_BIBLIOTHEQUE".Mobile[#index].Pos[0].Entr0_Ap_Pos[0] := "I_RPO_VPMP2_MLG2";
	"DB_BIBLIOTHEQUE".Mobile[#index].Pos[0].Entr1_Ap_Pos[0] := "I_RPF_VPMP2_MLG2";
	"DB_BIBLIOTHEQUE".Mobile[#index].Pos[0].Sort0[0] := "I_CO_VPMP2_MLG2";
	"DB_BIBLIOTHEQUE".Mobile[#index].Pos[0].Sort0_Pr_Fin_Pos[0] := "I_CO_VPMP2_MLG2";

	//position ouverture
	//Verouillage
	"DB_BIBLIOTHEQUE".Mobile[#index].Pos[1].Entr1_Av_Pos[0] := "I_RPF_VPMP2_MLG2";
	"DB_BIBLIOTHEQUE".Mobile[#index].Pos[1].Entr0_Ap_Pos[0] := "I_RPF_VPMP2_MLG2";
	"DB_BIBLIOTHEQUE".Mobile[#index].Pos[1].Entr1_Ap_Pos[0] := "I_RPO_VPMP2_MLG2";
	"DB_BIBLIOTHEQUE".Mobile[#index].Pos[1].Sort1[0] := "I_CO_VPMP2_MLG2";
	"DB_BIBLIOTHEQUE".Mobile[#index].Pos[1].Sort0_Pr_Fin_Pos[0] := "I_CO_VPMP2_MLG2";
	#index := #index + 1;
	//++++++++++++++++++++++++++++++++++++++++++++++++++++++++++++++/*340*/
	"DB_BIBLIOTHEQUE".Mobile[#index].Nom := 'VN3_MLG2';
	"DB_BIBLIOTHEQUE".Mobile[#index].Pos[0].Nom := 'FERMETURE';
	"DB_BIBLIOTHEQUE".Mobile[#index].Pos[1].Nom := 'OUVERTURE';
	"DB_BIBLIOTHEQUE".Mobile[#index].Tjr_Desasservi := TRUE;
	"Init_Tps"(#index);

	//position fermeture
	"DB_BIBLIOTHEQUE".Mobile[#index].Pos[0].Entr0_Ap_Pos[0] := "I_RPO_VPMP3_MLG2";
	"DB_BIBLIOTHEQUE".Mobile[#index].Pos[0].Entr1_Ap_Pos[0] := "I_RPF_VPMP3_MLG2";
	"DB_BIBLIOTHEQUE".Mobile[#index].Pos[0].Sort0[0] := "I_CO_VPMP3_MLG2";
	"DB_BIBLIOTHEQUE".Mobile[#index].Pos[0].Sort0_Pr_Fin_Pos[0] := "I_CO_VPMP3_MLG2";

	//position ouverture
	//Verouillage
	"DB_BIBLIOTHEQUE".Mobile[#index].Pos[1].Entr1_Av_Pos[0] := "I_RPF_VPMP3_MLG2";
	"DB_BIBLIOTHEQUE".Mobile[#index].Pos[1].Entr0_Ap_Pos[0] := "I_RPF_VPMP3_MLG2";
	"DB_BIBLIOTHEQUE".Mobile[#index].Pos[1].Entr1_Ap_Pos[0] := "I_RPO_VPMP3_MLG2";
	"DB_BIBLIOTHEQUE".Mobile[#index].Pos[1].Sort1[0] := "I_CO_VPMP3_MLG2";
	"DB_BIBLIOTHEQUE".Mobile[#index].Pos[1].Sort0_Pr_Fin_Pos[0] := "I_CO_VPMP3_MLG2";
	#index := #index + 1;
	//++++++++++++++++++++++++++++++++++++++++++++++++++++++++++++++/*341*/
	"DB_BIBLIOTHEQUE".Mobile[#index].Nom := 'VN4_MLG2';
	"DB_BIBLIOTHEQUE".Mobile[#index].Pos[0].Nom := 'FERMETURE';
	"DB_BIBLIOTHEQUE".Mobile[#index].Pos[1].Nom := 'OUVERTURE';
	"DB_BIBLIOTHEQUE".Mobile[#index].Tjr_Desasservi := TRUE;
	"Init_Tps"(#index);

	//position fermeture
	"DB_BIBLIOTHEQUE".Mobile[#index].Pos[0].Entr0_Ap_Pos[0] := "I_RPO_VPMP4_MLG2";
	"DB_BIBLIOTHEQUE".Mobile[#index].Pos[0].Entr1_Ap_Pos[0] := "I_RPF_VPMP4_MLG2";
	"DB_BIBLIOTHEQUE".Mobile[#index].Pos[0].Sort0[0] := "I_CO_VPMP4_MLG2";
	"DB_BIBLIOTHEQUE".Mobile[#index].Pos[0].Sort0_Pr_Fin_Pos[0] := "I_CO_VPMP4_MLG2";

	//position ouverture
	//Verouillage
	"DB_BIBLIOTHEQUE".Mobile[#index].Pos[1].Entr1_Av_Pos[0] := "I_RPF_VPMP4_MLG2";
	"DB_BIBLIOTHEQUE".Mobile[#index].Pos[1].Entr0_Ap_Pos[0] := "I_RPF_VPMP4_MLG2";
	"DB_BIBLIOTHEQUE".Mobile[#index].Pos[1].Entr1_Ap_Pos[0] := "I_RPO_VPMP4_MLG2";
	"DB_BIBLIOTHEQUE".Mobile[#index].Pos[1].Sort1[0] := "I_CO_VPMP4_MLG2";
	"DB_BIBLIOTHEQUE".Mobile[#index].Pos[1].Sort0_Pr_Fin_Pos[0] := "I_CO_VPMP4_MLG2";
	#index := #index + 1;
	//++++++++++++++++++++++++++++++++++++++++++++++++++++++++++++++/*342*/
	"DB_BIBLIOTHEQUE".Mobile[#index].Nom := 'VN5_MLG2';
	"DB_BIBLIOTHEQUE".Mobile[#index].Pos[0].Nom := 'FERMETURE';
	"DB_BIBLIOTHEQUE".Mobile[#index].Pos[1].Nom := 'OUVERTURE';
	"DB_BIBLIOTHEQUE".Mobile[#index].Tjr_Desasservi := TRUE;
	"Init_Tps"(#index);

	//position fermeture
	"DB_BIBLIOTHEQUE".Mobile[#index].Pos[0].Entr0_Ap_Pos[0] := "I_RPO_VPMP5_MLG2";
	"DB_BIBLIOTHEQUE".Mobile[#index].Pos[0].Entr1_Ap_Pos[0] := "I_RPF_VPMP5_MLG2";
	"DB_BIBLIOTHEQUE".Mobile[#index].Pos[0].Sort0[0] := "I_CO_VPMP5_MLG2";
	"DB_BIBLIOTHEQUE".Mobile[#index].Pos[0].Sort0_Pr_Fin_Pos[0] := "I_CO_VPMP5_MLG2";

	//position ouverture
	//Verouillage
	"DB_BIBLIOTHEQUE".Mobile[#index].Pos[1].Entr1_Av_Pos[0] := "I_RPF_VPMP5_MLG2";
	"DB_BIBLIOTHEQUE".Mobile[#index].Pos[1].Entr0_Ap_Pos[0] := "I_RPF_VPMP5_MLG2";
	"DB_BIBLIOTHEQUE".Mobile[#index].Pos[1].Entr1_Ap_Pos[0] := "I_RPO_VPMP5_MLG2";
	"DB_BIBLIOTHEQUE".Mobile[#index].Pos[1].Sort1[0] := "I_CO_VPMP5_MLG2";
	"DB_BIBLIOTHEQUE".Mobile[#index].Pos[1].Sort0_Pr_Fin_Pos[0] := "I_CO_VPMP5_MLG2";
	#index := #index + 1;
	//++++++++++++++++++++++++++++++++++++++++++++++++++++++++++++++/*343*/
	"DB_BIBLIOTHEQUE".Mobile[#index].Nom := 'TRP2_MLG1';
	"DB_BIBLIOTHEQUE".Mobile[#index].Pos[0].Nom := 'OUVERTURE';
	"DB_BIBLIOTHEQUE".Mobile[#index].Pos[1].Nom := 'FERMETURE';
	"DB_BIBLIOTHEQUE".Mobile[#index].Tjr_Desasservi := TRUE;
	"Init_Tps"(#index);

	// //position fermeture
	// "DB_BIBLIOTHEQUE".Mobile[#index].Pos[0].Entr0_Ap_Pos[0] := "I_RPO_TRP2_MLG";
	// "DB_BIBLIOTHEQUE".Mobile[#index].Pos[0].Entr1_Ap_Pos[0] := "I_RPF_TRP2_MLG";
	// "DB_BIBLIOTHEQUE".Mobile[#index].Pos[0].Sort0[0] := "I_CO_TRP2_MLG1";
	// "DB_BIBLIOTHEQUE".Mobile[#index].Pos[0].Sort0_Pr_Fin_Pos[0] := "I_CO_TRP2_MLG1";

	// //position ouverture
	// "DB_BIBLIOTHEQUE".Mobile[#index].Pos[1].Entr0_Ap_Pos[0] := "I_RPF_TRP2_MLG";
	// "DB_BIBLIOTHEQUE".Mobile[#index].Pos[1].Entr1_Ap_Pos[0] := "I_RPO_TRP2_MLG";
	// "DB_BIBLIOTHEQUE".Mobile[#index].Pos[1].Sort1[0] := "I_CO_TRP2_MLG1";
	// "DB_BIBLIOTHEQUE".Mobile[#index].Pos[1].Sort0_Pr_Fin_Pos[0] := "I_CO_TRP2_MLG1";
	#index := #index + 1;
	//++++++++++++++++++++++++++++++++++++++++++++++++++++++++++++++/*344*/
	"DB_BIBLIOTHEQUE".Mobile[#index].Nom := 'MLG2';
	"DB_BIBLIOTHEQUE".Mobile[#index].Pos[0].Nom := 'MARCHE';
	"DB_BIBLIOTHEQUE".Mobile[#index].Tjr_Desasservi := TRUE;
	"DB_BIBLIOTHEQUE".Mobile[#index].Tps_Att := t#500ms;
	"DB_BIBLIOTHEQUE".Mobile[#index].Tps_Arr := t#0ms;
	"DB_BIBLIOTHEQUE".Mobile[#index].Tps_Max_Mar_Forc := t#0ms;
	"DB_BIBLIOTHEQUE".Mobile[#index].Tps_Vid := t#0ms;

	// Entrées avant pos
	"DB_BIBLIOTHEQUE".Mobile[#index].Pos[0].Entr0_Av_Pos[0] := "I_RD_DISJ_MEL2";
	// Entrées apres pos
	"DB_BIBLIOTHEQUE".Mobile[#index].Pos[0].Entr0_Ap_Pos[0] := "I_RD_DISJ_MEL2";
	"DB_BIBLIOTHEQUE".Mobile[#index].Pos[0].Entr1_Ap_Pos[0] := "I_RM_MEL2";
	// Entrées fin pos
	"DB_BIBLIOTHEQUE".Mobile[#index].Pos[0].Entr0_Ap_Fin_Pos[0] := "I_RM_MEL2";
	// Sorties
	"DB_BIBLIOTHEQUE".Mobile[#index].Pos[0].Sort1[0] := "I_CM_MEL2";
	"DB_BIBLIOTHEQUE".Mobile[#index].Pos[0].Sort0_Pr_Fin_Pos[0] := "I_CM_MEL2";
	#index := #index + 1;
	//++++++++++++++++++++++++++++++++++++++++++++++++++++++++++++++/*345*/
	"DB_BIBLIOTHEQUE".Mobile[#index].Nom := 'TRP1_MLG2';
	"DB_BIBLIOTHEQUE".Mobile[#index].Pos[0].Nom := 'OUVERTURE';
	"DB_BIBLIOTHEQUE".Mobile[#index].Pos[1].Nom := 'FERMETURE';
	"DB_BIBLIOTHEQUE".Mobile[#index].Tjr_Desasservi := TRUE;
	"Init_Tps"(#index);

	//position fermeture
	"DB_BIBLIOTHEQUE".Mobile[#index].Pos[0].Entr0_Ap_Pos[0] := "I_RPO_TRP1_MLG2";
	"DB_BIBLIOTHEQUE".Mobile[#index].Pos[0].Entr1_Ap_Pos[0] := "I_RPF_TRP1_MLG2";
	"DB_BIBLIOTHEQUE".Mobile[#index].Pos[0].Sort0[0] := "I_CO_TRP1_MLG2";
	"DB_BIBLIOTHEQUE".Mobile[#index].Pos[0].Sort1_Pr_Fin_Pos[0] := "I_CO_TRP1_MLG2";
	//position fermeture
	"DB_BIBLIOTHEQUE".Mobile[#index].Pos[0].Entr0_Ap_Pos[1] := "I_RPO_TRP1_MLG2";
	"DB_BIBLIOTHEQUE".Mobile[#index].Pos[0].Entr1_Ap_Pos[1] := "I_RPF_TRP1_MLG2";
	"DB_BIBLIOTHEQUE".Mobile[#index].Pos[0].Sort0[1] := "I_CO_TRP1_MLG2";
	"DB_BIBLIOTHEQUE".Mobile[#index].Pos[0].Sort0_Pr_Fin_Pos[1] := "I_CO_TRP1_MLG2";

	//position ouverture
	"DB_BIBLIOTHEQUE".Mobile[#index].Pos[1].Entr0_Ap_Pos[0] := "I_RPF_TRP1_MLG2";
	"DB_BIBLIOTHEQUE".Mobile[#index].Pos[1].Entr1_Ap_Pos[0] := "I_RPO_TRP1_MLG2";
	"DB_BIBLIOTHEQUE".Mobile[#index].Pos[1].Sort1[0] := "I_CO_TRP1_MLG2";
	"DB_BIBLIOTHEQUE".Mobile[#index].Pos[1].Sort0_Pr_Fin_Pos[0] := "I_CO_TRP1_MLG2";
	//position ouverture
	"DB_BIBLIOTHEQUE".Mobile[#index].Pos[1].Entr0_Ap_Pos[1] := "I_RPF_TRP1_MLG2";
	"DB_BIBLIOTHEQUE".Mobile[#index].Pos[1].Entr1_Ap_Pos[1] := "I_RPO_TRP1_MLG2";
	"DB_BIBLIOTHEQUE".Mobile[#index].Pos[1].Sort1[1] := "I_CO_TRP1_MLG2";
	"DB_BIBLIOTHEQUE".Mobile[#index].Pos[1].Sort0_Pr_Fin_Pos[1] := "I_CO_TRP1_MLG2";
	#index := #index + 1;
	//++++++++++++++++++++++++++++++++++++++++++++++++++++++++++++++/*346*/
	"DB_BIBLIOTHEQUE".Mobile[#index].Nom := 'TRP2_MLG2';
	"DB_BIBLIOTHEQUE".Mobile[#index].Pos[0].Nom := 'OUVERTURE';
	"DB_BIBLIOTHEQUE".Mobile[#index].Pos[1].Nom := 'FERMETURE';
	"DB_BIBLIOTHEQUE".Mobile[#index].Tjr_Desasservi := TRUE;
	"Init_Tps"(#index);

